HMI tags "2905RS001A01F02"
   "2905RS001A01F02.MSW" : 52809b66-421d-457f-8884-6f7a49d4e247 AT %DB5024.DBX18.0, 500 ms
   "2905RS001A01F02.DefaultText" : TextRef, internal   // Заголовок POPUP окна. При експорте из ECS через скрипт заполняется автоматически, если теги копируются в ручную то требуется в ручную задатать свойство Start Value
   "2905RS001A01F02.BlockInfo" : Array [0..2] of Int AT %DB5024.DBX38.0, 500 ms
   "2905RS001A01F02.StatusWork" : Int AT %DB5024.DBW242, 500 ms
   "2905RS001A01F02.FP_PARAM.DampingTime" : Int AT %DB5024.DBW50, 500 ms
   "2905RS001A01F02.FP_PARAM.Force_Value" : Real AT %DB5024.DBD52, 500 ms
   "2905RS001A01F02.FP_PARAM.Scale_Min" : Real AT %DB5024.DBD56, 500 ms
   "2905RS001A01F02.FP_PARAM.Scale_Max" : Real AT %DB5024.DBD60, 500 ms
   "2905RS001A01F02.FP_PARAM.Gradient" : Real AT %DB5024.DBD64, 500 ms
   "2905RS001A01F02.FP_PARAM.Grad_Pos" : Real AT %DB5024.DBD68, 500 ms
   "2905RS001A01F02.FP_PARAM.Grad_Neg" : Real AT %DB5024.DBD72, 500 ms
   "2905RS001A01F02.FP_PARAM.Grad_X" : Real AT %DB5024.DBD76, 500 ms
   "2905RS001A01F02.FP_PARAM.Gradient_Time_Pre" : Int AT %DB5024.DBW80, 500 ms
   "2905RS001A01F02.FP_PARAM.Gradient_Time_ACC" : Int AT %DB5024.DBW82, 500 ms
   "2905RS001A01F02.FP_PARAM.Alarm_Hyst" : Real AT %DB5024.DBD84, 500 ms
   "2905RS001A01F02.FP_PARAM.AlarmLimit_H3" : Real AT %DB5024.DBD88, 500 ms
   "2905RS001A01F02.FP_PARAM.AlarmLimit_H2" : Real AT %DB5024.DBD92, 500 ms
   "2905RS001A01F02.FP_PARAM.AlarmLimit_H1" : Real AT %DB5024.DBD96, 500 ms
   "2905RS001A01F02.FP_PARAM.AlarmLimit_L1" : Real AT %DB5024.DBD100, 500 ms
   "2905RS001A01F02.FP_PARAM.AlarmLimit_L2" : Real AT %DB5024.DBD104, 500 ms
   "2905RS001A01F02.FP_PARAM.AlarmLimit_L3" : Real AT %DB5024.DBD108, 500 ms
   "2905RS001A01F02.FP_PARAM.AlarmDelay_H3_Pre" : Int AT %DB5024.DBW112, 500 ms
   "2905RS001A01F02.FP_PARAM.AlarmDelay_H3_Acc" : Int AT %DB5024.DBW114, 500 ms
   "2905RS001A01F02.FP_PARAM.AlarmDelay_H2_Pre" : Int AT %DB5024.DBW116, 500 ms
   "2905RS001A01F02.FP_PARAM.AlarmDelay_H2_Acc" : Int AT %DB5024.DBW118, 500 ms
   "2905RS001A01F02.FP_PARAM.AlarmDelay_H1_Pre" : Int AT %DB5024.DBW120, 500 ms
   "2905RS001A01F02.FP_PARAM.AlarmDelay_H1_Acc" : Int AT %DB5024.DBW122, 500 ms
   "2905RS001A01F02.FP_PARAM.AlarmDelay_L1_Pre" : Int AT %DB5024.DBW124, 500 ms
   "2905RS001A01F02.FP_PARAM.AlarmDelay_L1_Acc" : Int AT %DB5024.DBW126, 500 ms
   "2905RS001A01F02.FP_PARAM.AlarmDelay_L2_Pre" : Int AT %DB5024.DBW128, 500 ms
   "2905RS001A01F02.FP_PARAM.AlarmDelay_L2_Acc" : Int AT %DB5024.DBW130, 500 ms
   "2905RS001A01F02.FP_PARAM.AlarmDelay_L3_Pre" : Int AT %DB5024.DBW132, 500 ms
   "2905RS001A01F02.FP_PARAM.AlarmDelay_L3_Acc" : Int AT %DB5024.DBW134, 500 ms
   "2905RS001A01F02.FP_PARAM.OpenLoopDelay_Pre" : Int AT %DB5024.DBW136, 500 ms
   "2905RS001A01F02.FP_PARAM.OpenLoopDelay_Acc" : Int AT %DB5024.DBW138, 500 ms
   "2905RS001A01F02.FP_PARAM.OverRangeDelay_Pre" : Int AT %DB5024.DBW140, 500 ms
   "2905RS001A01F02.FP_PARAM.OverRangeDelay_Acc" : Int AT %DB5024.DBW142, 500 ms
   "2905RS001A01F02.FP_PARAM.AuxLimit_H2_Value" : Real AT %DB5024.DBD144, 500 ms
   "2905RS001A01F02.FP_PARAM.AuxLimit_H1_Value" : Real AT %DB5024.DBD148, 500 ms
   "2905RS001A01F02.FP_PARAM.AuxLimit_L2_Value" : Real AT %DB5024.DBD152, 500 ms
   "2905RS001A01F02.FP_PARAM.AuxLimit_L1_Value" : Real AT %DB5024.DBD156, 500 ms
   "2905RS001A01F02.Unit" : TextRef, internal   // Еденицы измерения При експорте из ECS через скрипт заполняется автоматически, если теги копируются в ручную то требуется задатать свойство Text
   "2905RS001A01F02.Decimals" : TextRef, internal   // Формат отображения При експорте из ECS через скрипт, заполняется автоматически. Если теги копируются в ручную то требуется задатать свойство Text s999999.9
   "2905RS001A01F02.FP_EN.Square" : Bool AT %DB5024.DBX46.0, 500 ms
   "2905RS001A01F02.FP_EN.SquareRoot" : Bool AT %DB5024.DBX46.1, 500 ms
   "2905RS001A01F02.FP_EN.ParentSupress" : Bool AT %DB5024.DBX46.2, 500 ms
   "2905RS001A01F02.FP_EN.ParentSupressUnit" : Bool AT %DB5024.DBX46.3, 500 ms
   "2905RS001A01F02.FP_EN.Force" : Bool AT %DB5024.DBX46.4, 500 ms
   "2905RS001A01F02.FP_EN.Damping" : Bool AT %DB5024.DBX46.5, 500 ms
   "2905RS001A01F02.FP_EN.Gradient_Pos" : Bool AT %DB5024.DBX46.6, 500 ms
   "2905RS001A01F02.FP_EN.Gradient_Neg" : Bool AT %DB5024.DBX46.7, 500 ms
   "2905RS001A01F02.FP_EN.Hysteresis" : Bool AT %DB5024.DBX47.0, 500 ms
   "2905RS001A01F02.FP_EN.Alarm_H3" : Bool AT %DB5024.DBX47.1, 500 ms
   "2905RS001A01F02.FP_EN.Alarm_H2" : Bool AT %DB5024.DBX47.2, 500 ms
   "2905RS001A01F02.FP_EN.Alarm_H1" : Bool AT %DB5024.DBX47.3, 500 ms
   "2905RS001A01F02.FP_EN.Alarm_L1" : Bool AT %DB5024.DBX47.4, 500 ms
   "2905RS001A01F02.FP_EN.Alarm_L2" : Bool AT %DB5024.DBX47.5, 500 ms
   "2905RS001A01F02.FP_EN.Alarm_L3" : Bool AT %DB5024.DBX47.6, 500 ms
   "2905RS001A01F02.FP_EN.AlarmDelay_H3" : Bool AT %DB5024.DBX47.7, 500 ms
   "2905RS001A01F02.FP_EN.AlarmDelay_H2" : Bool AT %DB5024.DBX48.0, 500 ms
   "2905RS001A01F02.FP_EN.AlarmDelay_H1" : Bool AT %DB5024.DBX48.1, 500 ms
   "2905RS001A01F02.FP_EN.AlarmDelay_L1" : Bool AT %DB5024.DBX48.2, 500 ms
   "2905RS001A01F02.FP_EN.AlarmDelay_L2" : Bool AT %DB5024.DBX48.3, 500 ms
   "2905RS001A01F02.FP_EN.AlarmDelay_L3" : Bool AT %DB5024.DBX48.4, 500 ms
   "2905RS001A01F02.FP_EN.ROC_Warn" : Bool AT %DB5024.DBX48.5, 500 ms
   "2905RS001A01F02.FP_EN.U_Range_Warn" : Bool AT %DB5024.DBX48.6, 500 ms
   "2905RS001A01F02.FP_EN.O_Range_Warn" : Bool AT %DB5024.DBX48.7, 500 ms
   "2905RS001A01F02.trend_tag_name" : TextRef, internal   // Еденицы измерения При експорте из ECS через скрипт - заполняется автоматически, если теги копируются в ручную то требуется задатать свойство Text - имя тега для тренда
   "2905RS001A01F02.DQ.AL_H3" : Bool AT %DB5024.DBX16.0, 500 ms
   "2905RS001A01F02.DQ.AL_H2" : Bool AT %DB5024.DBX16.1, 500 ms
   "2905RS001A01F02.DQ.AL_H1" : Bool AT %DB5024.DBX16.2, 500 ms
   "2905RS001A01F02.DQ.AL_L1" : Bool AT %DB5024.DBX16.3, 500 ms
   "2905RS001A01F02.DQ.AL_L2" : Bool AT %DB5024.DBX16.4, 500 ms
   "2905RS001A01F02.DQ.AL_L3" : Bool AT %DB5024.DBX16.5, 500 ms
   "2905RS001A01F02.DQ.SIG_OK" : Bool AT %DB5024.DBX16.6, 500 ms
   "2905RS001A01F02.DQ.LIM_H2" : Bool AT %DB5024.DBX16.7, 500 ms
   "2905RS001A01F02.DQ.LIM_H1" : Bool AT %DB5024.DBX17.0, 500 ms
   "2905RS001A01F02.DQ.LIM_L1" : Bool AT %DB5024.DBX17.1, 500 ms
   "2905RS001A01F02.DQ.LIM_L2" : Bool AT %DB5024.DBX17.2, 500 ms
   "2905RS001A01F02.DQ.GR_P" : Bool AT %DB5024.DBX17.3, 500 ms
   "2905RS001A01F02.DQ.GR_N" : Bool AT %DB5024.DBX17.4, 500 ms
   "2905RS001A01F02.I.IN" : Real AT %DB5024.DBD2, 500 ms
   "2905RS001A01F02.I.SIG_TYPE" : Int AT %DB5024.DBW0, 500 ms
   "2905RS001A01F02.I.FI_BUS" : Byte AT %DB5024.DBB6, 500 ms
   "2905RS001A01F02.DI.U_RANGE" : Bool AT %DB5024.DBX7.0, 500 ms
   "2905RS001A01F02.DI.O_RANGE" : Bool AT %DB5024.DBX7.1, 500 ms
   "2905RS001A01F02.DI.SIG_FAULT" : Bool AT %DB5024.DBX7.2, 500 ms
   "2905RS001A01F02.DI.EnConfig" : Bool AT %DB5024.DBX7.3, 500 ms
   "2905RS001A01F02.DI.AEN" : Bool AT %DB5024.DBX7.4, 500 ms
   "2905RS001A01F02.DI.AL_SUPR" : Bool AT %DB5024.DBX7.5, 500 ms
   "2905RS001A01F02.Q.PV_NORM" : Real AT %DB5024.DBD8, 500 ms
   "2905RS001A01F02.Q.PV_SCAL" : Real AT %DB5024.DBD12, 500 ms
   "2905RS001A01F02.ParentInfo" : TextRef, internal   // Имя родителя для попап окна, вкладка инфо. При експорте из ECS через скрипт заполняется автоматически, если теги копируются в ручную то требуется в ручную задатать свойство Start Value

HMI tags "2905RS001A01F03"
   "2905RS001A01F03.MSW" : 52809b66-421d-457f-8884-6f7a49d4e247 AT %DB5025.DBX18.0, 500 ms
   "2905RS001A01F03.DefaultText" : TextRef, internal   // Заголовок POPUP окна. При експорте из ECS через скрипт заполняется автоматически, если теги копируются в ручную то требуется в ручную задатать свойство Start Value
   "2905RS001A01F03.BlockInfo" : Array [0..2] of Int AT %DB5025.DBX38.0, 500 ms
   "2905RS001A01F03.StatusWork" : Int AT %DB5025.DBW242, 500 ms
   "2905RS001A01F03.FP_PARAM.DampingTime" : Int AT %DB5025.DBW50, 500 ms
   "2905RS001A01F03.FP_PARAM.Force_Value" : Real AT %DB5025.DBD52, 500 ms
   "2905RS001A01F03.FP_PARAM.Scale_Min" : Real AT %DB5025.DBD56, 500 ms
   "2905RS001A01F03.FP_PARAM.Scale_Max" : Real AT %DB5025.DBD60, 500 ms
   "2905RS001A01F03.FP_PARAM.Gradient" : Real AT %DB5025.DBD64, 500 ms
   "2905RS001A01F03.FP_PARAM.Grad_Pos" : Real AT %DB5025.DBD68, 500 ms
   "2905RS001A01F03.FP_PARAM.Grad_Neg" : Real AT %DB5025.DBD72, 500 ms
   "2905RS001A01F03.FP_PARAM.Grad_X" : Real AT %DB5025.DBD76, 500 ms
   "2905RS001A01F03.FP_PARAM.Gradient_Time_Pre" : Int AT %DB5025.DBW80, 500 ms
   "2905RS001A01F03.FP_PARAM.Gradient_Time_ACC" : Int AT %DB5025.DBW82, 500 ms
   "2905RS001A01F03.FP_PARAM.Alarm_Hyst" : Real AT %DB5025.DBD84, 500 ms
   "2905RS001A01F03.FP_PARAM.AlarmLimit_H3" : Real AT %DB5025.DBD88, 500 ms
   "2905RS001A01F03.FP_PARAM.AlarmLimit_H2" : Real AT %DB5025.DBD92, 500 ms
   "2905RS001A01F03.FP_PARAM.AlarmLimit_H1" : Real AT %DB5025.DBD96, 500 ms
   "2905RS001A01F03.FP_PARAM.AlarmLimit_L1" : Real AT %DB5025.DBD100, 500 ms
   "2905RS001A01F03.FP_PARAM.AlarmLimit_L2" : Real AT %DB5025.DBD104, 500 ms
   "2905RS001A01F03.FP_PARAM.AlarmLimit_L3" : Real AT %DB5025.DBD108, 500 ms
   "2905RS001A01F03.FP_PARAM.AlarmDelay_H3_Pre" : Int AT %DB5025.DBW112, 500 ms
   "2905RS001A01F03.FP_PARAM.AlarmDelay_H3_Acc" : Int AT %DB5025.DBW114, 500 ms
   "2905RS001A01F03.FP_PARAM.AlarmDelay_H2_Pre" : Int AT %DB5025.DBW116, 500 ms
   "2905RS001A01F03.FP_PARAM.AlarmDelay_H2_Acc" : Int AT %DB5025.DBW118, 500 ms
   "2905RS001A01F03.FP_PARAM.AlarmDelay_H1_Pre" : Int AT %DB5025.DBW120, 500 ms
   "2905RS001A01F03.FP_PARAM.AlarmDelay_H1_Acc" : Int AT %DB5025.DBW122, 500 ms
   "2905RS001A01F03.FP_PARAM.AlarmDelay_L1_Pre" : Int AT %DB5025.DBW124, 500 ms
   "2905RS001A01F03.FP_PARAM.AlarmDelay_L1_Acc" : Int AT %DB5025.DBW126, 500 ms
   "2905RS001A01F03.FP_PARAM.AlarmDelay_L2_Pre" : Int AT %DB5025.DBW128, 500 ms
   "2905RS001A01F03.FP_PARAM.AlarmDelay_L2_Acc" : Int AT %DB5025.DBW130, 500 ms
   "2905RS001A01F03.FP_PARAM.AlarmDelay_L3_Pre" : Int AT %DB5025.DBW132, 500 ms
   "2905RS001A01F03.FP_PARAM.AlarmDelay_L3_Acc" : Int AT %DB5025.DBW134, 500 ms
   "2905RS001A01F03.FP_PARAM.OpenLoopDelay_Pre" : Int AT %DB5025.DBW136, 500 ms
   "2905RS001A01F03.FP_PARAM.OpenLoopDelay_Acc" : Int AT %DB5025.DBW138, 500 ms
   "2905RS001A01F03.FP_PARAM.OverRangeDelay_Pre" : Int AT %DB5025.DBW140, 500 ms
   "2905RS001A01F03.FP_PARAM.OverRangeDelay_Acc" : Int AT %DB5025.DBW142, 500 ms
   "2905RS001A01F03.FP_PARAM.AuxLimit_H2_Value" : Real AT %DB5025.DBD144, 500 ms
   "2905RS001A01F03.FP_PARAM.AuxLimit_H1_Value" : Real AT %DB5025.DBD148, 500 ms
   "2905RS001A01F03.FP_PARAM.AuxLimit_L2_Value" : Real AT %DB5025.DBD152, 500 ms
   "2905RS001A01F03.FP_PARAM.AuxLimit_L1_Value" : Real AT %DB5025.DBD156, 500 ms
   "2905RS001A01F03.Unit" : TextRef, internal   // Еденицы измерения При експорте из ECS через скрипт заполняется автоматически, если теги копируются в ручную то требуется задатать свойство Text
   "2905RS001A01F03.Decimals" : TextRef, internal   // Формат отображения При експорте из ECS через скрипт, заполняется автоматически. Если теги копируются в ручную то требуется задатать свойство Text s999999.9
   "2905RS001A01F03.FP_EN.Square" : Bool AT %DB5025.DBX46.0, 500 ms
   "2905RS001A01F03.FP_EN.SquareRoot" : Bool AT %DB5025.DBX46.1, 500 ms
   "2905RS001A01F03.FP_EN.ParentSupress" : Bool AT %DB5025.DBX46.2, 500 ms
   "2905RS001A01F03.FP_EN.ParentSupressUnit" : Bool AT %DB5025.DBX46.3, 500 ms
   "2905RS001A01F03.FP_EN.Force" : Bool AT %DB5025.DBX46.4, 500 ms
   "2905RS001A01F03.FP_EN.Damping" : Bool AT %DB5025.DBX46.5, 500 ms
   "2905RS001A01F03.FP_EN.Gradient_Pos" : Bool AT %DB5025.DBX46.6, 500 ms
   "2905RS001A01F03.FP_EN.Gradient_Neg" : Bool AT %DB5025.DBX46.7, 500 ms
   "2905RS001A01F03.FP_EN.Hysteresis" : Bool AT %DB5025.DBX47.0, 500 ms
   "2905RS001A01F03.FP_EN.Alarm_H3" : Bool AT %DB5025.DBX47.1, 500 ms
   "2905RS001A01F03.FP_EN.Alarm_H2" : Bool AT %DB5025.DBX47.2, 500 ms
   "2905RS001A01F03.FP_EN.Alarm_H1" : Bool AT %DB5025.DBX47.3, 500 ms
   "2905RS001A01F03.FP_EN.Alarm_L1" : Bool AT %DB5025.DBX47.4, 500 ms
   "2905RS001A01F03.FP_EN.Alarm_L2" : Bool AT %DB5025.DBX47.5, 500 ms
   "2905RS001A01F03.FP_EN.Alarm_L3" : Bool AT %DB5025.DBX47.6, 500 ms
   "2905RS001A01F03.FP_EN.AlarmDelay_H3" : Bool AT %DB5025.DBX47.7, 500 ms
   "2905RS001A01F03.FP_EN.AlarmDelay_H2" : Bool AT %DB5025.DBX48.0, 500 ms
   "2905RS001A01F03.FP_EN.AlarmDelay_H1" : Bool AT %DB5025.DBX48.1, 500 ms
   "2905RS001A01F03.FP_EN.AlarmDelay_L1" : Bool AT %DB5025.DBX48.2, 500 ms
   "2905RS001A01F03.FP_EN.AlarmDelay_L2" : Bool AT %DB5025.DBX48.3, 500 ms
   "2905RS001A01F03.FP_EN.AlarmDelay_L3" : Bool AT %DB5025.DBX48.4, 500 ms
   "2905RS001A01F03.FP_EN.ROC_Warn" : Bool AT %DB5025.DBX48.5, 500 ms
   "2905RS001A01F03.FP_EN.U_Range_Warn" : Bool AT %DB5025.DBX48.6, 500 ms
   "2905RS001A01F03.FP_EN.O_Range_Warn" : Bool AT %DB5025.DBX48.7, 500 ms
   "2905RS001A01F03.trend_tag_name" : TextRef, internal   // Еденицы измерения При експорте из ECS через скрипт - заполняется автоматически, если теги копируются в ручную то требуется задатать свойство Text - имя тега для тренда
   "2905RS001A01F03.DQ.AL_H3" : Bool AT %DB5025.DBX16.0, 500 ms
   "2905RS001A01F03.DQ.AL_H2" : Bool AT %DB5025.DBX16.1, 500 ms
   "2905RS001A01F03.DQ.AL_H1" : Bool AT %DB5025.DBX16.2, 500 ms
   "2905RS001A01F03.DQ.AL_L1" : Bool AT %DB5025.DBX16.3, 500 ms
   "2905RS001A01F03.DQ.AL_L2" : Bool AT %DB5025.DBX16.4, 500 ms
   "2905RS001A01F03.DQ.AL_L3" : Bool AT %DB5025.DBX16.5, 500 ms
   "2905RS001A01F03.DQ.SIG_OK" : Bool AT %DB5025.DBX16.6, 500 ms
   "2905RS001A01F03.DQ.LIM_H2" : Bool AT %DB5025.DBX16.7, 500 ms
   "2905RS001A01F03.DQ.LIM_H1" : Bool AT %DB5025.DBX17.0, 500 ms
   "2905RS001A01F03.DQ.LIM_L1" : Bool AT %DB5025.DBX17.1, 500 ms
   "2905RS001A01F03.DQ.LIM_L2" : Bool AT %DB5025.DBX17.2, 500 ms
   "2905RS001A01F03.DQ.GR_P" : Bool AT %DB5025.DBX17.3, 500 ms
   "2905RS001A01F03.DQ.GR_N" : Bool AT %DB5025.DBX17.4, 500 ms
   "2905RS001A01F03.I.IN" : Real AT %DB5025.DBD2, 500 ms
   "2905RS001A01F03.I.SIG_TYPE" : Int AT %DB5025.DBW0, 500 ms
   "2905RS001A01F03.I.FI_BUS" : Byte AT %DB5025.DBB6, 500 ms
   "2905RS001A01F03.DI.U_RANGE" : Bool AT %DB5025.DBX7.0, 500 ms
   "2905RS001A01F03.DI.O_RANGE" : Bool AT %DB5025.DBX7.1, 500 ms
   "2905RS001A01F03.DI.SIG_FAULT" : Bool AT %DB5025.DBX7.2, 500 ms
   "2905RS001A01F03.DI.EnConfig" : Bool AT %DB5025.DBX7.3, 500 ms
   "2905RS001A01F03.DI.AEN" : Bool AT %DB5025.DBX7.4, 500 ms
   "2905RS001A01F03.DI.AL_SUPR" : Bool AT %DB5025.DBX7.5, 500 ms
   "2905RS001A01F03.Q.PV_NORM" : Real AT %DB5025.DBD8, 500 ms
   "2905RS001A01F03.Q.PV_SCAL" : Real AT %DB5025.DBD12, 500 ms
   "2905RS001A01F03.ParentInfo" : TextRef, internal   // Имя родителя для попап окна, вкладка инфо. При експорте из ECS через скрипт заполняется автоматически, если теги копируются в ручную то требуется в ручную задатать свойство Start Value

HMI tags "2905RS001A01F04"
   "2905RS001A01F04.MSW" : 52809b66-421d-457f-8884-6f7a49d4e247 AT %DB5026.DBX18.0, 500 ms
   "2905RS001A01F04.DefaultText" : TextRef, internal   // Заголовок POPUP окна. При експорте из ECS через скрипт заполняется автоматически, если теги копируются в ручную то требуется в ручную задатать свойство Start Value
   "2905RS001A01F04.BlockInfo" : Array [0..2] of Int AT %DB5026.DBX38.0, 500 ms
   "2905RS001A01F04.StatusWork" : Int AT %DB5026.DBW242, 500 ms
   "2905RS001A01F04.FP_PARAM.DampingTime" : Int AT %DB5026.DBW50, 500 ms
   "2905RS001A01F04.FP_PARAM.Force_Value" : Real AT %DB5026.DBD52, 500 ms
   "2905RS001A01F04.FP_PARAM.Scale_Min" : Real AT %DB5026.DBD56, 500 ms
   "2905RS001A01F04.FP_PARAM.Scale_Max" : Real AT %DB5026.DBD60, 500 ms
   "2905RS001A01F04.FP_PARAM.Gradient" : Real AT %DB5026.DBD64, 500 ms
   "2905RS001A01F04.FP_PARAM.Grad_Pos" : Real AT %DB5026.DBD68, 500 ms
   "2905RS001A01F04.FP_PARAM.Grad_Neg" : Real AT %DB5026.DBD72, 500 ms
   "2905RS001A01F04.FP_PARAM.Grad_X" : Real AT %DB5026.DBD76, 500 ms
   "2905RS001A01F04.FP_PARAM.Gradient_Time_Pre" : Int AT %DB5026.DBW80, 500 ms
   "2905RS001A01F04.FP_PARAM.Gradient_Time_ACC" : Int AT %DB5026.DBW82, 500 ms
   "2905RS001A01F04.FP_PARAM.Alarm_Hyst" : Real AT %DB5026.DBD84, 500 ms
   "2905RS001A01F04.FP_PARAM.AlarmLimit_H3" : Real AT %DB5026.DBD88, 500 ms
   "2905RS001A01F04.FP_PARAM.AlarmLimit_H2" : Real AT %DB5026.DBD92, 500 ms
   "2905RS001A01F04.FP_PARAM.AlarmLimit_H1" : Real AT %DB5026.DBD96, 500 ms
   "2905RS001A01F04.FP_PARAM.AlarmLimit_L1" : Real AT %DB5026.DBD100, 500 ms
   "2905RS001A01F04.FP_PARAM.AlarmLimit_L2" : Real AT %DB5026.DBD104, 500 ms
   "2905RS001A01F04.FP_PARAM.AlarmLimit_L3" : Real AT %DB5026.DBD108, 500 ms
   "2905RS001A01F04.FP_PARAM.AlarmDelay_H3_Pre" : Int AT %DB5026.DBW112, 500 ms
   "2905RS001A01F04.FP_PARAM.AlarmDelay_H3_Acc" : Int AT %DB5026.DBW114, 500 ms
   "2905RS001A01F04.FP_PARAM.AlarmDelay_H2_Pre" : Int AT %DB5026.DBW116, 500 ms
   "2905RS001A01F04.FP_PARAM.AlarmDelay_H2_Acc" : Int AT %DB5026.DBW118, 500 ms
   "2905RS001A01F04.FP_PARAM.AlarmDelay_H1_Pre" : Int AT %DB5026.DBW120, 500 ms
   "2905RS001A01F04.FP_PARAM.AlarmDelay_H1_Acc" : Int AT %DB5026.DBW122, 500 ms
   "2905RS001A01F04.FP_PARAM.AlarmDelay_L1_Pre" : Int AT %DB5026.DBW124, 500 ms
   "2905RS001A01F04.FP_PARAM.AlarmDelay_L1_Acc" : Int AT %DB5026.DBW126, 500 ms
   "2905RS001A01F04.FP_PARAM.AlarmDelay_L2_Pre" : Int AT %DB5026.DBW128, 500 ms
   "2905RS001A01F04.FP_PARAM.AlarmDelay_L2_Acc" : Int AT %DB5026.DBW130, 500 ms
   "2905RS001A01F04.FP_PARAM.AlarmDelay_L3_Pre" : Int AT %DB5026.DBW132, 500 ms
   "2905RS001A01F04.FP_PARAM.AlarmDelay_L3_Acc" : Int AT %DB5026.DBW134, 500 ms
   "2905RS001A01F04.FP_PARAM.OpenLoopDelay_Pre" : Int AT %DB5026.DBW136, 500 ms
   "2905RS001A01F04.FP_PARAM.OpenLoopDelay_Acc" : Int AT %DB5026.DBW138, 500 ms
   "2905RS001A01F04.FP_PARAM.OverRangeDelay_Pre" : Int AT %DB5026.DBW140, 500 ms
   "2905RS001A01F04.FP_PARAM.OverRangeDelay_Acc" : Int AT %DB5026.DBW142, 500 ms
   "2905RS001A01F04.FP_PARAM.AuxLimit_H2_Value" : Real AT %DB5026.DBD144, 500 ms
   "2905RS001A01F04.FP_PARAM.AuxLimit_H1_Value" : Real AT %DB5026.DBD148, 500 ms
   "2905RS001A01F04.FP_PARAM.AuxLimit_L2_Value" : Real AT %DB5026.DBD152, 500 ms
   "2905RS001A01F04.FP_PARAM.AuxLimit_L1_Value" : Real AT %DB5026.DBD156, 500 ms
   "2905RS001A01F04.Unit" : TextRef, internal   // Еденицы измерения При експорте из ECS через скрипт заполняется автоматически, если теги копируются в ручную то требуется задатать свойство Text
   "2905RS001A01F04.Decimals" : TextRef, internal   // Формат отображения При експорте из ECS через скрипт, заполняется автоматически. Если теги копируются в ручную то требуется задатать свойство Text s999999.9
   "2905RS001A01F04.FP_EN.Square" : Bool AT %DB5026.DBX46.0, 500 ms
   "2905RS001A01F04.FP_EN.SquareRoot" : Bool AT %DB5026.DBX46.1, 500 ms
   "2905RS001A01F04.FP_EN.ParentSupress" : Bool AT %DB5026.DBX46.2, 500 ms
   "2905RS001A01F04.FP_EN.ParentSupressUnit" : Bool AT %DB5026.DBX46.3, 500 ms
   "2905RS001A01F04.FP_EN.Force" : Bool AT %DB5026.DBX46.4, 500 ms
   "2905RS001A01F04.FP_EN.Damping" : Bool AT %DB5026.DBX46.5, 500 ms
   "2905RS001A01F04.FP_EN.Gradient_Pos" : Bool AT %DB5026.DBX46.6, 500 ms
   "2905RS001A01F04.FP_EN.Gradient_Neg" : Bool AT %DB5026.DBX46.7, 500 ms
   "2905RS001A01F04.FP_EN.Hysteresis" : Bool AT %DB5026.DBX47.0, 500 ms
   "2905RS001A01F04.FP_EN.Alarm_H3" : Bool AT %DB5026.DBX47.1, 500 ms
   "2905RS001A01F04.FP_EN.Alarm_H2" : Bool AT %DB5026.DBX47.2, 500 ms
   "2905RS001A01F04.FP_EN.Alarm_H1" : Bool AT %DB5026.DBX47.3, 500 ms
   "2905RS001A01F04.FP_EN.Alarm_L1" : Bool AT %DB5026.DBX47.4, 500 ms
   "2905RS001A01F04.FP_EN.Alarm_L2" : Bool AT %DB5026.DBX47.5, 500 ms
   "2905RS001A01F04.FP_EN.Alarm_L3" : Bool AT %DB5026.DBX47.6, 500 ms
   "2905RS001A01F04.FP_EN.AlarmDelay_H3" : Bool AT %DB5026.DBX47.7, 500 ms
   "2905RS001A01F04.FP_EN.AlarmDelay_H2" : Bool AT %DB5026.DBX48.0, 500 ms
   "2905RS001A01F04.FP_EN.AlarmDelay_H1" : Bool AT %DB5026.DBX48.1, 500 ms
   "2905RS001A01F04.FP_EN.AlarmDelay_L1" : Bool AT %DB5026.DBX48.2, 500 ms
   "2905RS001A01F04.FP_EN.AlarmDelay_L2" : Bool AT %DB5026.DBX48.3, 500 ms
   "2905RS001A01F04.FP_EN.AlarmDelay_L3" : Bool AT %DB5026.DBX48.4, 500 ms
   "2905RS001A01F04.FP_EN.ROC_Warn" : Bool AT %DB5026.DBX48.5, 500 ms
   "2905RS001A01F04.FP_EN.U_Range_Warn" : Bool AT %DB5026.DBX48.6, 500 ms
   "2905RS001A01F04.FP_EN.O_Range_Warn" : Bool AT %DB5026.DBX48.7, 500 ms
   "2905RS001A01F04.trend_tag_name" : TextRef, internal   // Еденицы измерения При експорте из ECS через скрипт - заполняется автоматически, если теги копируются в ручную то требуется задатать свойство Text - имя тега для тренда
   "2905RS001A01F04.DQ.AL_H3" : Bool AT %DB5026.DBX16.0, 500 ms
   "2905RS001A01F04.DQ.AL_H2" : Bool AT %DB5026.DBX16.1, 500 ms
   "2905RS001A01F04.DQ.AL_H1" : Bool AT %DB5026.DBX16.2, 500 ms
   "2905RS001A01F04.DQ.AL_L1" : Bool AT %DB5026.DBX16.3, 500 ms
   "2905RS001A01F04.DQ.AL_L2" : Bool AT %DB5026.DBX16.4, 500 ms
   "2905RS001A01F04.DQ.AL_L3" : Bool AT %DB5026.DBX16.5, 500 ms
   "2905RS001A01F04.DQ.SIG_OK" : Bool AT %DB5026.DBX16.6, 500 ms
   "2905RS001A01F04.DQ.LIM_H2" : Bool AT %DB5026.DBX16.7, 500 ms
   "2905RS001A01F04.DQ.LIM_H1" : Bool AT %DB5026.DBX17.0, 500 ms
   "2905RS001A01F04.DQ.LIM_L1" : Bool AT %DB5026.DBX17.1, 500 ms
   "2905RS001A01F04.DQ.LIM_L2" : Bool AT %DB5026.DBX17.2, 500 ms
   "2905RS001A01F04.DQ.GR_P" : Bool AT %DB5026.DBX17.3, 500 ms
   "2905RS001A01F04.DQ.GR_N" : Bool AT %DB5026.DBX17.4, 500 ms
   "2905RS001A01F04.I.IN" : Real AT %DB5026.DBD2, 500 ms
   "2905RS001A01F04.I.SIG_TYPE" : Int AT %DB5026.DBW0, 500 ms
   "2905RS001A01F04.I.FI_BUS" : Byte AT %DB5026.DBB6, 500 ms
   "2905RS001A01F04.DI.U_RANGE" : Bool AT %DB5026.DBX7.0, 500 ms
   "2905RS001A01F04.DI.O_RANGE" : Bool AT %DB5026.DBX7.1, 500 ms
   "2905RS001A01F04.DI.SIG_FAULT" : Bool AT %DB5026.DBX7.2, 500 ms
   "2905RS001A01F04.DI.EnConfig" : Bool AT %DB5026.DBX7.3, 500 ms
   "2905RS001A01F04.DI.AEN" : Bool AT %DB5026.DBX7.4, 500 ms
   "2905RS001A01F04.DI.AL_SUPR" : Bool AT %DB5026.DBX7.5, 500 ms
   "2905RS001A01F04.Q.PV_NORM" : Real AT %DB5026.DBD8, 500 ms
   "2905RS001A01F04.Q.PV_SCAL" : Real AT %DB5026.DBD12, 500 ms
   "2905RS001A01F04.ParentInfo" : TextRef, internal   // Имя родителя для попап окна, вкладка инфо. При експорте из ECS через скрипт заполняется автоматически, если теги копируются в ручную то требуется в ручную задатать свойство Start Value

HMI tags "2905RS001A01L01"
   "2905RS001A01L01.MSW" : 52809b66-421d-457f-8884-6f7a49d4e247 AT %DB5027.DBX18.0, 500 ms
   "2905RS001A01L01.DefaultText" : TextRef, internal   // Заголовок POPUP окна. При експорте из ECS через скрипт заполняется автоматически, если теги копируются в ручную то требуется в ручную задатать свойство Start Value
   "2905RS001A01L01.BlockInfo" : Array [0..2] of Int AT %DB5027.DBX38.0, 500 ms
   "2905RS001A01L01.StatusWork" : Int AT %DB5027.DBW242, 500 ms
   "2905RS001A01L01.FP_PARAM.DampingTime" : Int AT %DB5027.DBW50, 500 ms
   "2905RS001A01L01.FP_PARAM.Force_Value" : Real AT %DB5027.DBD52, 500 ms
   "2905RS001A01L01.FP_PARAM.Scale_Min" : Real AT %DB5027.DBD56, 500 ms
   "2905RS001A01L01.FP_PARAM.Scale_Max" : Real AT %DB5027.DBD60, 500 ms
   "2905RS001A01L01.FP_PARAM.Gradient" : Real AT %DB5027.DBD64, 500 ms
   "2905RS001A01L01.FP_PARAM.Grad_Pos" : Real AT %DB5027.DBD68, 500 ms
   "2905RS001A01L01.FP_PARAM.Grad_Neg" : Real AT %DB5027.DBD72, 500 ms
   "2905RS001A01L01.FP_PARAM.Grad_X" : Real AT %DB5027.DBD76, 500 ms
   "2905RS001A01L01.FP_PARAM.Gradient_Time_Pre" : Int AT %DB5027.DBW80, 500 ms
   "2905RS001A01L01.FP_PARAM.Gradient_Time_ACC" : Int AT %DB5027.DBW82, 500 ms
   "2905RS001A01L01.FP_PARAM.Alarm_Hyst" : Real AT %DB5027.DBD84, 500 ms
   "2905RS001A01L01.FP_PARAM.AlarmLimit_H3" : Real AT %DB5027.DBD88, 500 ms
   "2905RS001A01L01.FP_PARAM.AlarmLimit_H2" : Real AT %DB5027.DBD92, 500 ms
   "2905RS001A01L01.FP_PARAM.AlarmLimit_H1" : Real AT %DB5027.DBD96, 500 ms
   "2905RS001A01L01.FP_PARAM.AlarmLimit_L1" : Real AT %DB5027.DBD100, 500 ms
   "2905RS001A01L01.FP_PARAM.AlarmLimit_L2" : Real AT %DB5027.DBD104, 500 ms
   "2905RS001A01L01.FP_PARAM.AlarmLimit_L3" : Real AT %DB5027.DBD108, 500 ms
   "2905RS001A01L01.FP_PARAM.AlarmDelay_H3_Pre" : Int AT %DB5027.DBW112, 500 ms
   "2905RS001A01L01.FP_PARAM.AlarmDelay_H3_Acc" : Int AT %DB5027.DBW114, 500 ms
   "2905RS001A01L01.FP_PARAM.AlarmDelay_H2_Pre" : Int AT %DB5027.DBW116, 500 ms
   "2905RS001A01L01.FP_PARAM.AlarmDelay_H2_Acc" : Int AT %DB5027.DBW118, 500 ms
   "2905RS001A01L01.FP_PARAM.AlarmDelay_H1_Pre" : Int AT %DB5027.DBW120, 500 ms
   "2905RS001A01L01.FP_PARAM.AlarmDelay_H1_Acc" : Int AT %DB5027.DBW122, 500 ms
   "2905RS001A01L01.FP_PARAM.AlarmDelay_L1_Pre" : Int AT %DB5027.DBW124, 500 ms
   "2905RS001A01L01.FP_PARAM.AlarmDelay_L1_Acc" : Int AT %DB5027.DBW126, 500 ms
   "2905RS001A01L01.FP_PARAM.AlarmDelay_L2_Pre" : Int AT %DB5027.DBW128, 500 ms
   "2905RS001A01L01.FP_PARAM.AlarmDelay_L2_Acc" : Int AT %DB5027.DBW130, 500 ms
   "2905RS001A01L01.FP_PARAM.AlarmDelay_L3_Pre" : Int AT %DB5027.DBW132, 500 ms
   "2905RS001A01L01.FP_PARAM.AlarmDelay_L3_Acc" : Int AT %DB5027.DBW134, 500 ms
   "2905RS001A01L01.FP_PARAM.OpenLoopDelay_Pre" : Int AT %DB5027.DBW136, 500 ms
   "2905RS001A01L01.FP_PARAM.OpenLoopDelay_Acc" : Int AT %DB5027.DBW138, 500 ms
   "2905RS001A01L01.FP_PARAM.OverRangeDelay_Pre" : Int AT %DB5027.DBW140, 500 ms
   "2905RS001A01L01.FP_PARAM.OverRangeDelay_Acc" : Int AT %DB5027.DBW142, 500 ms
   "2905RS001A01L01.FP_PARAM.AuxLimit_H2_Value" : Real AT %DB5027.DBD144, 500 ms
   "2905RS001A01L01.FP_PARAM.AuxLimit_H1_Value" : Real AT %DB5027.DBD148, 500 ms
   "2905RS001A01L01.FP_PARAM.AuxLimit_L2_Value" : Real AT %DB5027.DBD152, 500 ms
   "2905RS001A01L01.FP_PARAM.AuxLimit_L1_Value" : Real AT %DB5027.DBD156, 500 ms
   "2905RS001A01L01.Unit" : TextRef, internal   // Еденицы измерения При експорте из ECS через скрипт заполняется автоматически, если теги копируются в ручную то требуется задатать свойство Text
   "2905RS001A01L01.Decimals" : TextRef, internal   // Формат отображения При експорте из ECS через скрипт, заполняется автоматически. Если теги копируются в ручную то требуется задатать свойство Text s999999.9
   "2905RS001A01L01.FP_EN.Square" : Bool AT %DB5027.DBX46.0, 500 ms
   "2905RS001A01L01.FP_EN.SquareRoot" : Bool AT %DB5027.DBX46.1, 500 ms
   "2905RS001A01L01.FP_EN.ParentSupress" : Bool AT %DB5027.DBX46.2, 500 ms
   "2905RS001A01L01.FP_EN.ParentSupressUnit" : Bool AT %DB5027.DBX46.3, 500 ms
   "2905RS001A01L01.FP_EN.Force" : Bool AT %DB5027.DBX46.4, 500 ms
   "2905RS001A01L01.FP_EN.Damping" : Bool AT %DB5027.DBX46.5, 500 ms
   "2905RS001A01L01.FP_EN.Gradient_Pos" : Bool AT %DB5027.DBX46.6, 500 ms
   "2905RS001A01L01.FP_EN.Gradient_Neg" : Bool AT %DB5027.DBX46.7, 500 ms
   "2905RS001A01L01.FP_EN.Hysteresis" : Bool AT %DB5027.DBX47.0, 500 ms
   "2905RS001A01L01.FP_EN.Alarm_H3" : Bool AT %DB5027.DBX47.1, 500 ms
   "2905RS001A01L01.FP_EN.Alarm_H2" : Bool AT %DB5027.DBX47.2, 500 ms
   "2905RS001A01L01.FP_EN.Alarm_H1" : Bool AT %DB5027.DBX47.3, 500 ms
   "2905RS001A01L01.FP_EN.Alarm_L1" : Bool AT %DB5027.DBX47.4, 500 ms
   "2905RS001A01L01.FP_EN.Alarm_L2" : Bool AT %DB5027.DBX47.5, 500 ms
   "2905RS001A01L01.FP_EN.Alarm_L3" : Bool AT %DB5027.DBX47.6, 500 ms
   "2905RS001A01L01.FP_EN.AlarmDelay_H3" : Bool AT %DB5027.DBX47.7, 500 ms
   "2905RS001A01L01.FP_EN.AlarmDelay_H2" : Bool AT %DB5027.DBX48.0, 500 ms
   "2905RS001A01L01.FP_EN.AlarmDelay_H1" : Bool AT %DB5027.DBX48.1, 500 ms
   "2905RS001A01L01.FP_EN.AlarmDelay_L1" : Bool AT %DB5027.DBX48.2, 500 ms
   "2905RS001A01L01.FP_EN.AlarmDelay_L2" : Bool AT %DB5027.DBX48.3, 500 ms
   "2905RS001A01L01.FP_EN.AlarmDelay_L3" : Bool AT %DB5027.DBX48.4, 500 ms
   "2905RS001A01L01.FP_EN.ROC_Warn" : Bool AT %DB5027.DBX48.5, 500 ms
   "2905RS001A01L01.FP_EN.U_Range_Warn" : Bool AT %DB5027.DBX48.6, 500 ms
   "2905RS001A01L01.FP_EN.O_Range_Warn" : Bool AT %DB5027.DBX48.7, 500 ms
   "2905RS001A01L01.trend_tag_name" : TextRef, internal   // Еденицы измерения При експорте из ECS через скрипт - заполняется автоматически, если теги копируются в ручную то требуется задатать свойство Text - имя тега для тренда
   "2905RS001A01L01.DQ.AL_H3" : Bool AT %DB5027.DBX16.0, 500 ms
   "2905RS001A01L01.DQ.AL_H2" : Bool AT %DB5027.DBX16.1, 500 ms
   "2905RS001A01L01.DQ.AL_H1" : Bool AT %DB5027.DBX16.2, 500 ms
   "2905RS001A01L01.DQ.AL_L1" : Bool AT %DB5027.DBX16.3, 500 ms
   "2905RS001A01L01.DQ.AL_L2" : Bool AT %DB5027.DBX16.4, 500 ms
   "2905RS001A01L01.DQ.AL_L3" : Bool AT %DB5027.DBX16.5, 500 ms
   "2905RS001A01L01.DQ.SIG_OK" : Bool AT %DB5027.DBX16.6, 500 ms
   "2905RS001A01L01.DQ.LIM_H2" : Bool AT %DB5027.DBX16.7, 500 ms
   "2905RS001A01L01.DQ.LIM_H1" : Bool AT %DB5027.DBX17.0, 500 ms
   "2905RS001A01L01.DQ.LIM_L1" : Bool AT %DB5027.DBX17.1, 500 ms
   "2905RS001A01L01.DQ.LIM_L2" : Bool AT %DB5027.DBX17.2, 500 ms
   "2905RS001A01L01.DQ.GR_P" : Bool AT %DB5027.DBX17.3, 500 ms
   "2905RS001A01L01.DQ.GR_N" : Bool AT %DB5027.DBX17.4, 500 ms
   "2905RS001A01L01.I.IN" : Real AT %DB5027.DBD2, 500 ms
   "2905RS001A01L01.I.SIG_TYPE" : Int AT %DB5027.DBW0, 500 ms
   "2905RS001A01L01.I.FI_BUS" : Byte AT %DB5027.DBB6, 500 ms
   "2905RS001A01L01.DI.U_RANGE" : Bool AT %DB5027.DBX7.0, 500 ms
   "2905RS001A01L01.DI.O_RANGE" : Bool AT %DB5027.DBX7.1, 500 ms
   "2905RS001A01L01.DI.SIG_FAULT" : Bool AT %DB5027.DBX7.2, 500 ms
   "2905RS001A01L01.DI.EnConfig" : Bool AT %DB5027.DBX7.3, 500 ms
   "2905RS001A01L01.DI.AEN" : Bool AT %DB5027.DBX7.4, 500 ms
   "2905RS001A01L01.DI.AL_SUPR" : Bool AT %DB5027.DBX7.5, 500 ms
   "2905RS001A01L01.Q.PV_NORM" : Real AT %DB5027.DBD8, 500 ms
   "2905RS001A01L01.Q.PV_SCAL" : Real AT %DB5027.DBD12, 500 ms
   "2905RS001A01L01.ParentInfo" : TextRef, internal   // Имя родителя для попап окна, вкладка инфо. При експорте из ECS через скрипт заполняется автоматически, если теги копируются в ручную то требуется в ручную задатать свойство Start Value

HMI tags "2910RS001A01F01"
   "2910RS001A01F01.MSW" : 52809b66-421d-457f-8884-6f7a49d4e247 AT %DB5030.DBX18.0, 500 ms
   "2910RS001A01F01.DefaultText" : TextRef, internal   // Заголовок POPUP окна. При експорте из ECS через скрипт заполняется автоматически, если теги копируются в ручную то требуется в ручную задатать свойство Start Value
   "2910RS001A01F01.BlockInfo" : Array [0..2] of Int AT %DB5030.DBX38.0, 500 ms
   "2910RS001A01F01.StatusWork" : Int AT %DB5030.DBW242, 500 ms
   "2910RS001A01F01.FP_PARAM.DampingTime" : Int AT %DB5030.DBW50, 500 ms
   "2910RS001A01F01.FP_PARAM.Force_Value" : Real AT %DB5030.DBD52, 500 ms
   "2910RS001A01F01.FP_PARAM.Scale_Min" : Real AT %DB5030.DBD56, 500 ms
   "2910RS001A01F01.FP_PARAM.Scale_Max" : Real AT %DB5030.DBD60, 500 ms
   "2910RS001A01F01.FP_PARAM.Gradient" : Real AT %DB5030.DBD64, 500 ms
   "2910RS001A01F01.FP_PARAM.Grad_Pos" : Real AT %DB5030.DBD68, 500 ms
   "2910RS001A01F01.FP_PARAM.Grad_Neg" : Real AT %DB5030.DBD72, 500 ms
   "2910RS001A01F01.FP_PARAM.Grad_X" : Real AT %DB5030.DBD76, 500 ms
   "2910RS001A01F01.FP_PARAM.Gradient_Time_Pre" : Int AT %DB5030.DBW80, 500 ms
   "2910RS001A01F01.FP_PARAM.Gradient_Time_ACC" : Int AT %DB5030.DBW82, 500 ms
   "2910RS001A01F01.FP_PARAM.Alarm_Hyst" : Real AT %DB5030.DBD84, 500 ms
   "2910RS001A01F01.FP_PARAM.AlarmLimit_H3" : Real AT %DB5030.DBD88, 500 ms
   "2910RS001A01F01.FP_PARAM.AlarmLimit_H2" : Real AT %DB5030.DBD92, 500 ms
   "2910RS001A01F01.FP_PARAM.AlarmLimit_H1" : Real AT %DB5030.DBD96, 500 ms
   "2910RS001A01F01.FP_PARAM.AlarmLimit_L1" : Real AT %DB5030.DBD100, 500 ms
   "2910RS001A01F01.FP_PARAM.AlarmLimit_L2" : Real AT %DB5030.DBD104, 500 ms
   "2910RS001A01F01.FP_PARAM.AlarmLimit_L3" : Real AT %DB5030.DBD108, 500 ms
   "2910RS001A01F01.FP_PARAM.AlarmDelay_H3_Pre" : Int AT %DB5030.DBW112, 500 ms
   "2910RS001A01F01.FP_PARAM.AlarmDelay_H3_Acc" : Int AT %DB5030.DBW114, 500 ms
   "2910RS001A01F01.FP_PARAM.AlarmDelay_H2_Pre" : Int AT %DB5030.DBW116, 500 ms
   "2910RS001A01F01.FP_PARAM.AlarmDelay_H2_Acc" : Int AT %DB5030.DBW118, 500 ms
   "2910RS001A01F01.FP_PARAM.AlarmDelay_H1_Pre" : Int AT %DB5030.DBW120, 500 ms
   "2910RS001A01F01.FP_PARAM.AlarmDelay_H1_Acc" : Int AT %DB5030.DBW122, 500 ms
   "2910RS001A01F01.FP_PARAM.AlarmDelay_L1_Pre" : Int AT %DB5030.DBW124, 500 ms
   "2910RS001A01F01.FP_PARAM.AlarmDelay_L1_Acc" : Int AT %DB5030.DBW126, 500 ms
   "2910RS001A01F01.FP_PARAM.AlarmDelay_L2_Pre" : Int AT %DB5030.DBW128, 500 ms
   "2910RS001A01F01.FP_PARAM.AlarmDelay_L2_Acc" : Int AT %DB5030.DBW130, 500 ms
   "2910RS001A01F01.FP_PARAM.AlarmDelay_L3_Pre" : Int AT %DB5030.DBW132, 500 ms
   "2910RS001A01F01.FP_PARAM.AlarmDelay_L3_Acc" : Int AT %DB5030.DBW134, 500 ms
   "2910RS001A01F01.FP_PARAM.OpenLoopDelay_Pre" : Int AT %DB5030.DBW136, 500 ms
   "2910RS001A01F01.FP_PARAM.OpenLoopDelay_Acc" : Int AT %DB5030.DBW138, 500 ms
   "2910RS001A01F01.FP_PARAM.OverRangeDelay_Pre" : Int AT %DB5030.DBW140, 500 ms
   "2910RS001A01F01.FP_PARAM.OverRangeDelay_Acc" : Int AT %DB5030.DBW142, 500 ms
   "2910RS001A01F01.FP_PARAM.AuxLimit_H2_Value" : Real AT %DB5030.DBD144, 500 ms
   "2910RS001A01F01.FP_PARAM.AuxLimit_H1_Value" : Real AT %DB5030.DBD148, 500 ms
   "2910RS001A01F01.FP_PARAM.AuxLimit_L2_Value" : Real AT %DB5030.DBD152, 500 ms
   "2910RS001A01F01.FP_PARAM.AuxLimit_L1_Value" : Real AT %DB5030.DBD156, 500 ms
   "2910RS001A01F01.Unit" : TextRef, internal   // Еденицы измерения При експорте из ECS через скрипт заполняется автоматически, если теги копируются в ручную то требуется задатать свойство Text
   "2910RS001A01F01.Decimals" : TextRef, internal   // Формат отображения При експорте из ECS через скрипт, заполняется автоматически. Если теги копируются в ручную то требуется задатать свойство Text s999999.9
   "2910RS001A01F01.FP_EN.Square" : Bool AT %DB5030.DBX46.0, 500 ms
   "2910RS001A01F01.FP_EN.SquareRoot" : Bool AT %DB5030.DBX46.1, 500 ms
   "2910RS001A01F01.FP_EN.ParentSupress" : Bool AT %DB5030.DBX46.2, 500 ms
   "2910RS001A01F01.FP_EN.ParentSupressUnit" : Bool AT %DB5030.DBX46.3, 500 ms
   "2910RS001A01F01.FP_EN.Force" : Bool AT %DB5030.DBX46.4, 500 ms
   "2910RS001A01F01.FP_EN.Damping" : Bool AT %DB5030.DBX46.5, 500 ms
   "2910RS001A01F01.FP_EN.Gradient_Pos" : Bool AT %DB5030.DBX46.6, 500 ms
   "2910RS001A01F01.FP_EN.Gradient_Neg" : Bool AT %DB5030.DBX46.7, 500 ms
   "2910RS001A01F01.FP_EN.Hysteresis" : Bool AT %DB5030.DBX47.0, 500 ms
   "2910RS001A01F01.FP_EN.Alarm_H3" : Bool AT %DB5030.DBX47.1, 500 ms
   "2910RS001A01F01.FP_EN.Alarm_H2" : Bool AT %DB5030.DBX47.2, 500 ms
   "2910RS001A01F01.FP_EN.Alarm_H1" : Bool AT %DB5030.DBX47.3, 500 ms
   "2910RS001A01F01.FP_EN.Alarm_L1" : Bool AT %DB5030.DBX47.4, 500 ms
   "2910RS001A01F01.FP_EN.Alarm_L2" : Bool AT %DB5030.DBX47.5, 500 ms
   "2910RS001A01F01.FP_EN.Alarm_L3" : Bool AT %DB5030.DBX47.6, 500 ms
   "2910RS001A01F01.FP_EN.AlarmDelay_H3" : Bool AT %DB5030.DBX47.7, 500 ms
   "2910RS001A01F01.FP_EN.AlarmDelay_H2" : Bool AT %DB5030.DBX48.0, 500 ms
   "2910RS001A01F01.FP_EN.AlarmDelay_H1" : Bool AT %DB5030.DBX48.1, 500 ms
   "2910RS001A01F01.FP_EN.AlarmDelay_L1" : Bool AT %DB5030.DBX48.2, 500 ms
   "2910RS001A01F01.FP_EN.AlarmDelay_L2" : Bool AT %DB5030.DBX48.3, 500 ms
   "2910RS001A01F01.FP_EN.AlarmDelay_L3" : Bool AT %DB5030.DBX48.4, 500 ms
   "2910RS001A01F01.FP_EN.ROC_Warn" : Bool AT %DB5030.DBX48.5, 500 ms
   "2910RS001A01F01.FP_EN.U_Range_Warn" : Bool AT %DB5030.DBX48.6, 500 ms
   "2910RS001A01F01.FP_EN.O_Range_Warn" : Bool AT %DB5030.DBX48.7, 500 ms
   "2910RS001A01F01.trend_tag_name" : TextRef, internal   // Еденицы измерения При експорте из ECS через скрипт - заполняется автоматически, если теги копируются в ручную то требуется задатать свойство Text - имя тега для тренда
   "2910RS001A01F01.DQ.AL_H3" : Bool AT %DB5030.DBX16.0, 500 ms
   "2910RS001A01F01.DQ.AL_H2" : Bool AT %DB5030.DBX16.1, 500 ms
   "2910RS001A01F01.DQ.AL_H1" : Bool AT %DB5030.DBX16.2, 500 ms
   "2910RS001A01F01.DQ.AL_L1" : Bool AT %DB5030.DBX16.3, 500 ms
   "2910RS001A01F01.DQ.AL_L2" : Bool AT %DB5030.DBX16.4, 500 ms
   "2910RS001A01F01.DQ.AL_L3" : Bool AT %DB5030.DBX16.5, 500 ms
   "2910RS001A01F01.DQ.SIG_OK" : Bool AT %DB5030.DBX16.6, 500 ms
   "2910RS001A01F01.DQ.LIM_H2" : Bool AT %DB5030.DBX16.7, 500 ms
   "2910RS001A01F01.DQ.LIM_H1" : Bool AT %DB5030.DBX17.0, 500 ms
   "2910RS001A01F01.DQ.LIM_L1" : Bool AT %DB5030.DBX17.1, 500 ms
   "2910RS001A01F01.DQ.LIM_L2" : Bool AT %DB5030.DBX17.2, 500 ms
   "2910RS001A01F01.DQ.GR_P" : Bool AT %DB5030.DBX17.3, 500 ms
   "2910RS001A01F01.DQ.GR_N" : Bool AT %DB5030.DBX17.4, 500 ms
   "2910RS001A01F01.I.IN" : Real AT %DB5030.DBD2, 500 ms
   "2910RS001A01F01.I.SIG_TYPE" : Int AT %DB5030.DBW0, 500 ms
   "2910RS001A01F01.I.FI_BUS" : Byte AT %DB5030.DBB6, 500 ms
   "2910RS001A01F01.DI.U_RANGE" : Bool AT %DB5030.DBX7.0, 500 ms
   "2910RS001A01F01.DI.O_RANGE" : Bool AT %DB5030.DBX7.1, 500 ms
   "2910RS001A01F01.DI.SIG_FAULT" : Bool AT %DB5030.DBX7.2, 500 ms
   "2910RS001A01F01.DI.EnConfig" : Bool AT %DB5030.DBX7.3, 500 ms
   "2910RS001A01F01.DI.AEN" : Bool AT %DB5030.DBX7.4, 500 ms
   "2910RS001A01F01.DI.AL_SUPR" : Bool AT %DB5030.DBX7.5, 500 ms
   "2910RS001A01F01.Q.PV_NORM" : Real AT %DB5030.DBD8, 500 ms
   "2910RS001A01F01.Q.PV_SCAL" : Real AT %DB5030.DBD12, 500 ms
   "2910RS001A01F01.ParentInfo" : TextRef, internal   // Имя родителя для попап окна, вкладка инфо. При експорте из ECS через скрипт заполняется автоматически, если теги копируются в ручную то требуется в ручную задатать свойство Start Value

HMI tags "2910RS001A01L01"
   "2910RS001A01L01.MSW" : 52809b66-421d-457f-8884-6f7a49d4e247 AT %DB5031.DBX18.0, 500 ms
   "2910RS001A01L01.DefaultText" : TextRef, internal   // Заголовок POPUP окна. При експорте из ECS через скрипт заполняется автоматически, если теги копируются в ручную то требуется в ручную задатать свойство Start Value
   "2910RS001A01L01.BlockInfo" : Array [0..2] of Int AT %DB5031.DBX38.0, 500 ms
   "2910RS001A01L01.StatusWork" : Int AT %DB5031.DBW242, 500 ms
   "2910RS001A01L01.FP_PARAM.DampingTime" : Int AT %DB5031.DBW50, 500 ms
   "2910RS001A01L01.FP_PARAM.Force_Value" : Real AT %DB5031.DBD52, 500 ms
   "2910RS001A01L01.FP_PARAM.Scale_Min" : Real AT %DB5031.DBD56, 500 ms
   "2910RS001A01L01.FP_PARAM.Scale_Max" : Real AT %DB5031.DBD60, 500 ms
   "2910RS001A01L01.FP_PARAM.Gradient" : Real AT %DB5031.DBD64, 500 ms
   "2910RS001A01L01.FP_PARAM.Grad_Pos" : Real AT %DB5031.DBD68, 500 ms
   "2910RS001A01L01.FP_PARAM.Grad_Neg" : Real AT %DB5031.DBD72, 500 ms
   "2910RS001A01L01.FP_PARAM.Grad_X" : Real AT %DB5031.DBD76, 500 ms
   "2910RS001A01L01.FP_PARAM.Gradient_Time_Pre" : Int AT %DB5031.DBW80, 500 ms
   "2910RS001A01L01.FP_PARAM.Gradient_Time_ACC" : Int AT %DB5031.DBW82, 500 ms
   "2910RS001A01L01.FP_PARAM.Alarm_Hyst" : Real AT %DB5031.DBD84, 500 ms
   "2910RS001A01L01.FP_PARAM.AlarmLimit_H3" : Real AT %DB5031.DBD88, 500 ms
   "2910RS001A01L01.FP_PARAM.AlarmLimit_H2" : Real AT %DB5031.DBD92, 500 ms
   "2910RS001A01L01.FP_PARAM.AlarmLimit_H1" : Real AT %DB5031.DBD96, 500 ms
   "2910RS001A01L01.FP_PARAM.AlarmLimit_L1" : Real AT %DB5031.DBD100, 500 ms
   "2910RS001A01L01.FP_PARAM.AlarmLimit_L2" : Real AT %DB5031.DBD104, 500 ms
   "2910RS001A01L01.FP_PARAM.AlarmLimit_L3" : Real AT %DB5031.DBD108, 500 ms
   "2910RS001A01L01.FP_PARAM.AlarmDelay_H3_Pre" : Int AT %DB5031.DBW112, 500 ms
   "2910RS001A01L01.FP_PARAM.AlarmDelay_H3_Acc" : Int AT %DB5031.DBW114, 500 ms
   "2910RS001A01L01.FP_PARAM.AlarmDelay_H2_Pre" : Int AT %DB5031.DBW116, 500 ms
   "2910RS001A01L01.FP_PARAM.AlarmDelay_H2_Acc" : Int AT %DB5031.DBW118, 500 ms
   "2910RS001A01L01.FP_PARAM.AlarmDelay_H1_Pre" : Int AT %DB5031.DBW120, 500 ms
   "2910RS001A01L01.FP_PARAM.AlarmDelay_H1_Acc" : Int AT %DB5031.DBW122, 500 ms
   "2910RS001A01L01.FP_PARAM.AlarmDelay_L1_Pre" : Int AT %DB5031.DBW124, 500 ms
   "2910RS001A01L01.FP_PARAM.AlarmDelay_L1_Acc" : Int AT %DB5031.DBW126, 500 ms
   "2910RS001A01L01.FP_PARAM.AlarmDelay_L2_Pre" : Int AT %DB5031.DBW128, 500 ms
   "2910RS001A01L01.FP_PARAM.AlarmDelay_L2_Acc" : Int AT %DB5031.DBW130, 500 ms
   "2910RS001A01L01.FP_PARAM.AlarmDelay_L3_Pre" : Int AT %DB5031.DBW132, 500 ms
   "2910RS001A01L01.FP_PARAM.AlarmDelay_L3_Acc" : Int AT %DB5031.DBW134, 500 ms
   "2910RS001A01L01.FP_PARAM.OpenLoopDelay_Pre" : Int AT %DB5031.DBW136, 500 ms
   "2910RS001A01L01.FP_PARAM.OpenLoopDelay_Acc" : Int AT %DB5031.DBW138, 500 ms
   "2910RS001A01L01.FP_PARAM.OverRangeDelay_Pre" : Int AT %DB5031.DBW140, 500 ms
   "2910RS001A01L01.FP_PARAM.OverRangeDelay_Acc" : Int AT %DB5031.DBW142, 500 ms
   "2910RS001A01L01.FP_PARAM.AuxLimit_H2_Value" : Real AT %DB5031.DBD144, 500 ms
   "2910RS001A01L01.FP_PARAM.AuxLimit_H1_Value" : Real AT %DB5031.DBD148, 500 ms
   "2910RS001A01L01.FP_PARAM.AuxLimit_L2_Value" : Real AT %DB5031.DBD152, 500 ms
   "2910RS001A01L01.FP_PARAM.AuxLimit_L1_Value" : Real AT %DB5031.DBD156, 500 ms
   "2910RS001A01L01.Unit" : TextRef, internal   // Еденицы измерения При експорте из ECS через скрипт заполняется автоматически, если теги копируются в ручную то требуется задатать свойство Text
   "2910RS001A01L01.Decimals" : TextRef, internal   // Формат отображения При експорте из ECS через скрипт, заполняется автоматически. Если теги копируются в ручную то требуется задатать свойство Text s999999.9
   "2910RS001A01L01.FP_EN.Square" : Bool AT %DB5031.DBX46.0, 500 ms
   "2910RS001A01L01.FP_EN.SquareRoot" : Bool AT %DB5031.DBX46.1, 500 ms
   "2910RS001A01L01.FP_EN.ParentSupress" : Bool AT %DB5031.DBX46.2, 500 ms
   "2910RS001A01L01.FP_EN.ParentSupressUnit" : Bool AT %DB5031.DBX46.3, 500 ms
   "2910RS001A01L01.FP_EN.Force" : Bool AT %DB5031.DBX46.4, 500 ms
   "2910RS001A01L01.FP_EN.Damping" : Bool AT %DB5031.DBX46.5, 500 ms
   "2910RS001A01L01.FP_EN.Gradient_Pos" : Bool AT %DB5031.DBX46.6, 500 ms
   "2910RS001A01L01.FP_EN.Gradient_Neg" : Bool AT %DB5031.DBX46.7, 500 ms
   "2910RS001A01L01.FP_EN.Hysteresis" : Bool AT %DB5031.DBX47.0, 500 ms
   "2910RS001A01L01.FP_EN.Alarm_H3" : Bool AT %DB5031.DBX47.1, 500 ms
   "2910RS001A01L01.FP_EN.Alarm_H2" : Bool AT %DB5031.DBX47.2, 500 ms
   "2910RS001A01L01.FP_EN.Alarm_H1" : Bool AT %DB5031.DBX47.3, 500 ms
   "2910RS001A01L01.FP_EN.Alarm_L1" : Bool AT %DB5031.DBX47.4, 500 ms
   "2910RS001A01L01.FP_EN.Alarm_L2" : Bool AT %DB5031.DBX47.5, 500 ms
   "2910RS001A01L01.FP_EN.Alarm_L3" : Bool AT %DB5031.DBX47.6, 500 ms
   "2910RS001A01L01.FP_EN.AlarmDelay_H3" : Bool AT %DB5031.DBX47.7, 500 ms
   "2910RS001A01L01.FP_EN.AlarmDelay_H2" : Bool AT %DB5031.DBX48.0, 500 ms
   "2910RS001A01L01.FP_EN.AlarmDelay_H1" : Bool AT %DB5031.DBX48.1, 500 ms
   "2910RS001A01L01.FP_EN.AlarmDelay_L1" : Bool AT %DB5031.DBX48.2, 500 ms
   "2910RS001A01L01.FP_EN.AlarmDelay_L2" : Bool AT %DB5031.DBX48.3, 500 ms
   "2910RS001A01L01.FP_EN.AlarmDelay_L3" : Bool AT %DB5031.DBX48.4, 500 ms
   "2910RS001A01L01.FP_EN.ROC_Warn" : Bool AT %DB5031.DBX48.5, 500 ms
   "2910RS001A01L01.FP_EN.U_Range_Warn" : Bool AT %DB5031.DBX48.6, 500 ms
   "2910RS001A01L01.FP_EN.O_Range_Warn" : Bool AT %DB5031.DBX48.7, 500 ms
   "2910RS001A01L01.trend_tag_name" : TextRef, internal   // Еденицы измерения При експорте из ECS через скрипт - заполняется автоматически, если теги копируются в ручную то требуется задатать свойство Text - имя тега для тренда
   "2910RS001A01L01.DQ.AL_H3" : Bool AT %DB5031.DBX16.0, 500 ms
   "2910RS001A01L01.DQ.AL_H2" : Bool AT %DB5031.DBX16.1, 500 ms
   "2910RS001A01L01.DQ.AL_H1" : Bool AT %DB5031.DBX16.2, 500 ms
   "2910RS001A01L01.DQ.AL_L1" : Bool AT %DB5031.DBX16.3, 500 ms
   "2910RS001A01L01.DQ.AL_L2" : Bool AT %DB5031.DBX16.4, 500 ms
   "2910RS001A01L01.DQ.AL_L3" : Bool AT %DB5031.DBX16.5, 500 ms
   "2910RS001A01L01.DQ.SIG_OK" : Bool AT %DB5031.DBX16.6, 500 ms
   "2910RS001A01L01.DQ.LIM_H2" : Bool AT %DB5031.DBX16.7, 500 ms
   "2910RS001A01L01.DQ.LIM_H1" : Bool AT %DB5031.DBX17.0, 500 ms
   "2910RS001A01L01.DQ.LIM_L1" : Bool AT %DB5031.DBX17.1, 500 ms
   "2910RS001A01L01.DQ.LIM_L2" : Bool AT %DB5031.DBX17.2, 500 ms
   "2910RS001A01L01.DQ.GR_P" : Bool AT %DB5031.DBX17.3, 500 ms
   "2910RS001A01L01.DQ.GR_N" : Bool AT %DB5031.DBX17.4, 500 ms
   "2910RS001A01L01.I.IN" : Real AT %DB5031.DBD2, 500 ms
   "2910RS001A01L01.I.SIG_TYPE" : Int AT %DB5031.DBW0, 500 ms
   "2910RS001A01L01.I.FI_BUS" : Byte AT %DB5031.DBB6, 500 ms
   "2910RS001A01L01.DI.U_RANGE" : Bool AT %DB5031.DBX7.0, 500 ms
   "2910RS001A01L01.DI.O_RANGE" : Bool AT %DB5031.DBX7.1, 500 ms
   "2910RS001A01L01.DI.SIG_FAULT" : Bool AT %DB5031.DBX7.2, 500 ms
   "2910RS001A01L01.DI.EnConfig" : Bool AT %DB5031.DBX7.3, 500 ms
   "2910RS001A01L01.DI.AEN" : Bool AT %DB5031.DBX7.4, 500 ms
   "2910RS001A01L01.DI.AL_SUPR" : Bool AT %DB5031.DBX7.5, 500 ms
   "2910RS001A01L01.Q.PV_NORM" : Real AT %DB5031.DBD8, 500 ms
   "2910RS001A01L01.Q.PV_SCAL" : Real AT %DB5031.DBD12, 500 ms
   "2910RS001A01L01.ParentInfo" : TextRef, internal   // Имя родителя для попап окна, вкладка инфо. При експорте из ECS через скрипт заполняется автоматически, если теги копируются в ручную то требуется в ручную задатать свойство Start Value

HMI tags "2910RS001A01L02"
   "2910RS001A01L02.MSW" : 52809b66-421d-457f-8884-6f7a49d4e247 AT %DB5032.DBX18.0, 500 ms
   "2910RS001A01L02.DefaultText" : TextRef, internal   // Заголовок POPUP окна. При експорте из ECS через скрипт заполняется автоматически, если теги копируются в ручную то требуется в ручную задатать свойство Start Value
   "2910RS001A01L02.BlockInfo" : Array [0..2] of Int AT %DB5032.DBX38.0, 500 ms
   "2910RS001A01L02.StatusWork" : Int AT %DB5032.DBW242, 500 ms
   "2910RS001A01L02.FP_PARAM.DampingTime" : Int AT %DB5032.DBW50, 500 ms
   "2910RS001A01L02.FP_PARAM.Force_Value" : Real AT %DB5032.DBD52, 500 ms
   "2910RS001A01L02.FP_PARAM.Scale_Min" : Real AT %DB5032.DBD56, 500 ms
   "2910RS001A01L02.FP_PARAM.Scale_Max" : Real AT %DB5032.DBD60, 500 ms
   "2910RS001A01L02.FP_PARAM.Gradient" : Real AT %DB5032.DBD64, 500 ms
   "2910RS001A01L02.FP_PARAM.Grad_Pos" : Real AT %DB5032.DBD68, 500 ms
   "2910RS001A01L02.FP_PARAM.Grad_Neg" : Real AT %DB5032.DBD72, 500 ms
   "2910RS001A01L02.FP_PARAM.Grad_X" : Real AT %DB5032.DBD76, 500 ms
   "2910RS001A01L02.FP_PARAM.Gradient_Time_Pre" : Int AT %DB5032.DBW80, 500 ms
   "2910RS001A01L02.FP_PARAM.Gradient_Time_ACC" : Int AT %DB5032.DBW82, 500 ms
   "2910RS001A01L02.FP_PARAM.Alarm_Hyst" : Real AT %DB5032.DBD84, 500 ms
   "2910RS001A01L02.FP_PARAM.AlarmLimit_H3" : Real AT %DB5032.DBD88, 500 ms
   "2910RS001A01L02.FP_PARAM.AlarmLimit_H2" : Real AT %DB5032.DBD92, 500 ms
   "2910RS001A01L02.FP_PARAM.AlarmLimit_H1" : Real AT %DB5032.DBD96, 500 ms
   "2910RS001A01L02.FP_PARAM.AlarmLimit_L1" : Real AT %DB5032.DBD100, 500 ms
   "2910RS001A01L02.FP_PARAM.AlarmLimit_L2" : Real AT %DB5032.DBD104, 500 ms
   "2910RS001A01L02.FP_PARAM.AlarmLimit_L3" : Real AT %DB5032.DBD108, 500 ms
   "2910RS001A01L02.FP_PARAM.AlarmDelay_H3_Pre" : Int AT %DB5032.DBW112, 500 ms
   "2910RS001A01L02.FP_PARAM.AlarmDelay_H3_Acc" : Int AT %DB5032.DBW114, 500 ms
   "2910RS001A01L02.FP_PARAM.AlarmDelay_H2_Pre" : Int AT %DB5032.DBW116, 500 ms
   "2910RS001A01L02.FP_PARAM.AlarmDelay_H2_Acc" : Int AT %DB5032.DBW118, 500 ms
   "2910RS001A01L02.FP_PARAM.AlarmDelay_H1_Pre" : Int AT %DB5032.DBW120, 500 ms
   "2910RS001A01L02.FP_PARAM.AlarmDelay_H1_Acc" : Int AT %DB5032.DBW122, 500 ms
   "2910RS001A01L02.FP_PARAM.AlarmDelay_L1_Pre" : Int AT %DB5032.DBW124, 500 ms
   "2910RS001A01L02.FP_PARAM.AlarmDelay_L1_Acc" : Int AT %DB5032.DBW126, 500 ms
   "2910RS001A01L02.FP_PARAM.AlarmDelay_L2_Pre" : Int AT %DB5032.DBW128, 500 ms
   "2910RS001A01L02.FP_PARAM.AlarmDelay_L2_Acc" : Int AT %DB5032.DBW130, 500 ms
   "2910RS001A01L02.FP_PARAM.AlarmDelay_L3_Pre" : Int AT %DB5032.DBW132, 500 ms
   "2910RS001A01L02.FP_PARAM.AlarmDelay_L3_Acc" : Int AT %DB5032.DBW134, 500 ms
   "2910RS001A01L02.FP_PARAM.OpenLoopDelay_Pre" : Int AT %DB5032.DBW136, 500 ms
   "2910RS001A01L02.FP_PARAM.OpenLoopDelay_Acc" : Int AT %DB5032.DBW138, 500 ms
   "2910RS001A01L02.FP_PARAM.OverRangeDelay_Pre" : Int AT %DB5032.DBW140, 500 ms
   "2910RS001A01L02.FP_PARAM.OverRangeDelay_Acc" : Int AT %DB5032.DBW142, 500 ms
   "2910RS001A01L02.FP_PARAM.AuxLimit_H2_Value" : Real AT %DB5032.DBD144, 500 ms
   "2910RS001A01L02.FP_PARAM.AuxLimit_H1_Value" : Real AT %DB5032.DBD148, 500 ms
   "2910RS001A01L02.FP_PARAM.AuxLimit_L2_Value" : Real AT %DB5032.DBD152, 500 ms
   "2910RS001A01L02.FP_PARAM.AuxLimit_L1_Value" : Real AT %DB5032.DBD156, 500 ms
   "2910RS001A01L02.Unit" : TextRef, internal   // Еденицы измерения При експорте из ECS через скрипт заполняется автоматически, если теги копируются в ручную то требуется задатать свойство Text
   "2910RS001A01L02.Decimals" : TextRef, internal   // Формат отображения При експорте из ECS через скрипт, заполняется автоматически. Если теги копируются в ручную то требуется задатать свойство Text s999999.9
   "2910RS001A01L02.FP_EN.Square" : Bool AT %DB5032.DBX46.0, 500 ms
   "2910RS001A01L02.FP_EN.SquareRoot" : Bool AT %DB5032.DBX46.1, 500 ms
   "2910RS001A01L02.FP_EN.ParentSupress" : Bool AT %DB5032.DBX46.2, 500 ms
   "2910RS001A01L02.FP_EN.ParentSupressUnit" : Bool AT %DB5032.DBX46.3, 500 ms
   "2910RS001A01L02.FP_EN.Force" : Bool AT %DB5032.DBX46.4, 500 ms
   "2910RS001A01L02.FP_EN.Damping" : Bool AT %DB5032.DBX46.5, 500 ms
   "2910RS001A01L02.FP_EN.Gradient_Pos" : Bool AT %DB5032.DBX46.6, 500 ms
   "2910RS001A01L02.FP_EN.Gradient_Neg" : Bool AT %DB5032.DBX46.7, 500 ms
   "2910RS001A01L02.FP_EN.Hysteresis" : Bool AT %DB5032.DBX47.0, 500 ms
   "2910RS001A01L02.FP_EN.Alarm_H3" : Bool AT %DB5032.DBX47.1, 500 ms
   "2910RS001A01L02.FP_EN.Alarm_H2" : Bool AT %DB5032.DBX47.2, 500 ms
   "2910RS001A01L02.FP_EN.Alarm_H1" : Bool AT %DB5032.DBX47.3, 500 ms
   "2910RS001A01L02.FP_EN.Alarm_L1" : Bool AT %DB5032.DBX47.4, 500 ms
   "2910RS001A01L02.FP_EN.Alarm_L2" : Bool AT %DB5032.DBX47.5, 500 ms
   "2910RS001A01L02.FP_EN.Alarm_L3" : Bool AT %DB5032.DBX47.6, 500 ms
   "2910RS001A01L02.FP_EN.AlarmDelay_H3" : Bool AT %DB5032.DBX47.7, 500 ms
   "2910RS001A01L02.FP_EN.AlarmDelay_H2" : Bool AT %DB5032.DBX48.0, 500 ms
   "2910RS001A01L02.FP_EN.AlarmDelay_H1" : Bool AT %DB5032.DBX48.1, 500 ms
   "2910RS001A01L02.FP_EN.AlarmDelay_L1" : Bool AT %DB5032.DBX48.2, 500 ms
   "2910RS001A01L02.FP_EN.AlarmDelay_L2" : Bool AT %DB5032.DBX48.3, 500 ms
   "2910RS001A01L02.FP_EN.AlarmDelay_L3" : Bool AT %DB5032.DBX48.4, 500 ms
   "2910RS001A01L02.FP_EN.ROC_Warn" : Bool AT %DB5032.DBX48.5, 500 ms
   "2910RS001A01L02.FP_EN.U_Range_Warn" : Bool AT %DB5032.DBX48.6, 500 ms
   "2910RS001A01L02.FP_EN.O_Range_Warn" : Bool AT %DB5032.DBX48.7, 500 ms
   "2910RS001A01L02.trend_tag_name" : TextRef, internal   // Еденицы измерения При експорте из ECS через скрипт - заполняется автоматически, если теги копируются в ручную то требуется задатать свойство Text - имя тега для тренда
   "2910RS001A01L02.DQ.AL_H3" : Bool AT %DB5032.DBX16.0, 500 ms
   "2910RS001A01L02.DQ.AL_H2" : Bool AT %DB5032.DBX16.1, 500 ms
   "2910RS001A01L02.DQ.AL_H1" : Bool AT %DB5032.DBX16.2, 500 ms
   "2910RS001A01L02.DQ.AL_L1" : Bool AT %DB5032.DBX16.3, 500 ms
   "2910RS001A01L02.DQ.AL_L2" : Bool AT %DB5032.DBX16.4, 500 ms
   "2910RS001A01L02.DQ.AL_L3" : Bool AT %DB5032.DBX16.5, 500 ms
   "2910RS001A01L02.DQ.SIG_OK" : Bool AT %DB5032.DBX16.6, 500 ms
   "2910RS001A01L02.DQ.LIM_H2" : Bool AT %DB5032.DBX16.7, 500 ms
   "2910RS001A01L02.DQ.LIM_H1" : Bool AT %DB5032.DBX17.0, 500 ms
   "2910RS001A01L02.DQ.LIM_L1" : Bool AT %DB5032.DBX17.1, 500 ms
   "2910RS001A01L02.DQ.LIM_L2" : Bool AT %DB5032.DBX17.2, 500 ms
   "2910RS001A01L02.DQ.GR_P" : Bool AT %DB5032.DBX17.3, 500 ms
   "2910RS001A01L02.DQ.GR_N" : Bool AT %DB5032.DBX17.4, 500 ms
   "2910RS001A01L02.I.IN" : Real AT %DB5032.DBD2, 500 ms
   "2910RS001A01L02.I.SIG_TYPE" : Int AT %DB5032.DBW0, 500 ms
   "2910RS001A01L02.I.FI_BUS" : Byte AT %DB5032.DBB6, 500 ms
   "2910RS001A01L02.DI.U_RANGE" : Bool AT %DB5032.DBX7.0, 500 ms
   "2910RS001A01L02.DI.O_RANGE" : Bool AT %DB5032.DBX7.1, 500 ms
   "2910RS001A01L02.DI.SIG_FAULT" : Bool AT %DB5032.DBX7.2, 500 ms
   "2910RS001A01L02.DI.EnConfig" : Bool AT %DB5032.DBX7.3, 500 ms
   "2910RS001A01L02.DI.AEN" : Bool AT %DB5032.DBX7.4, 500 ms
   "2910RS001A01L02.DI.AL_SUPR" : Bool AT %DB5032.DBX7.5, 500 ms
   "2910RS001A01L02.Q.PV_NORM" : Real AT %DB5032.DBD8, 500 ms
   "2910RS001A01L02.Q.PV_SCAL" : Real AT %DB5032.DBD12, 500 ms
   "2910RS001A01L02.ParentInfo" : TextRef, internal   // Имя родителя для попап окна, вкладка инфо. При експорте из ECS через скрипт заполняется автоматически, если теги копируются в ручную то требуется в ручную задатать свойство Start Value

HMI tags "2910RS001A01N01"
   "2910RS001A01N01.MSW" : 52809b66-421d-457f-8884-6f7a49d4e247 AT %DB5033.DBX18.0, 500 ms
   "2910RS001A01N01.DefaultText" : TextRef, internal   // Заголовок POPUP окна. При експорте из ECS через скрипт заполняется автоматически, если теги копируются в ручную то требуется в ручную задатать свойство Start Value
   "2910RS001A01N01.BlockInfo" : Array [0..2] of Int AT %DB5033.DBX38.0, 500 ms
   "2910RS001A01N01.StatusWork" : Int AT %DB5033.DBW242, 500 ms
   "2910RS001A01N01.FP_PARAM.DampingTime" : Int AT %DB5033.DBW50, 500 ms
   "2910RS001A01N01.FP_PARAM.Force_Value" : Real AT %DB5033.DBD52, 500 ms
   "2910RS001A01N01.FP_PARAM.Scale_Min" : Real AT %DB5033.DBD56, 500 ms
   "2910RS001A01N01.FP_PARAM.Scale_Max" : Real AT %DB5033.DBD60, 500 ms
   "2910RS001A01N01.FP_PARAM.Gradient" : Real AT %DB5033.DBD64, 500 ms
   "2910RS001A01N01.FP_PARAM.Grad_Pos" : Real AT %DB5033.DBD68, 500 ms
   "2910RS001A01N01.FP_PARAM.Grad_Neg" : Real AT %DB5033.DBD72, 500 ms
   "2910RS001A01N01.FP_PARAM.Grad_X" : Real AT %DB5033.DBD76, 500 ms
   "2910RS001A01N01.FP_PARAM.Gradient_Time_Pre" : Int AT %DB5033.DBW80, 500 ms
   "2910RS001A01N01.FP_PARAM.Gradient_Time_ACC" : Int AT %DB5033.DBW82, 500 ms
   "2910RS001A01N01.FP_PARAM.Alarm_Hyst" : Real AT %DB5033.DBD84, 500 ms
   "2910RS001A01N01.FP_PARAM.AlarmLimit_H3" : Real AT %DB5033.DBD88, 500 ms
   "2910RS001A01N01.FP_PARAM.AlarmLimit_H2" : Real AT %DB5033.DBD92, 500 ms
   "2910RS001A01N01.FP_PARAM.AlarmLimit_H1" : Real AT %DB5033.DBD96, 500 ms
   "2910RS001A01N01.FP_PARAM.AlarmLimit_L1" : Real AT %DB5033.DBD100, 500 ms
   "2910RS001A01N01.FP_PARAM.AlarmLimit_L2" : Real AT %DB5033.DBD104, 500 ms
   "2910RS001A01N01.FP_PARAM.AlarmLimit_L3" : Real AT %DB5033.DBD108, 500 ms
   "2910RS001A01N01.FP_PARAM.AlarmDelay_H3_Pre" : Int AT %DB5033.DBW112, 500 ms
   "2910RS001A01N01.FP_PARAM.AlarmDelay_H3_Acc" : Int AT %DB5033.DBW114, 500 ms
   "2910RS001A01N01.FP_PARAM.AlarmDelay_H2_Pre" : Int AT %DB5033.DBW116, 500 ms
   "2910RS001A01N01.FP_PARAM.AlarmDelay_H2_Acc" : Int AT %DB5033.DBW118, 500 ms
   "2910RS001A01N01.FP_PARAM.AlarmDelay_H1_Pre" : Int AT %DB5033.DBW120, 500 ms
   "2910RS001A01N01.FP_PARAM.AlarmDelay_H1_Acc" : Int AT %DB5033.DBW122, 500 ms
   "2910RS001A01N01.FP_PARAM.AlarmDelay_L1_Pre" : Int AT %DB5033.DBW124, 500 ms
   "2910RS001A01N01.FP_PARAM.AlarmDelay_L1_Acc" : Int AT %DB5033.DBW126, 500 ms
   "2910RS001A01N01.FP_PARAM.AlarmDelay_L2_Pre" : Int AT %DB5033.DBW128, 500 ms
   "2910RS001A01N01.FP_PARAM.AlarmDelay_L2_Acc" : Int AT %DB5033.DBW130, 500 ms
   "2910RS001A01N01.FP_PARAM.AlarmDelay_L3_Pre" : Int AT %DB5033.DBW132, 500 ms
   "2910RS001A01N01.FP_PARAM.AlarmDelay_L3_Acc" : Int AT %DB5033.DBW134, 500 ms
   "2910RS001A01N01.FP_PARAM.OpenLoopDelay_Pre" : Int AT %DB5033.DBW136, 500 ms
   "2910RS001A01N01.FP_PARAM.OpenLoopDelay_Acc" : Int AT %DB5033.DBW138, 500 ms
   "2910RS001A01N01.FP_PARAM.OverRangeDelay_Pre" : Int AT %DB5033.DBW140, 500 ms
   "2910RS001A01N01.FP_PARAM.OverRangeDelay_Acc" : Int AT %DB5033.DBW142, 500 ms
   "2910RS001A01N01.FP_PARAM.AuxLimit_H2_Value" : Real AT %DB5033.DBD144, 500 ms
   "2910RS001A01N01.FP_PARAM.AuxLimit_H1_Value" : Real AT %DB5033.DBD148, 500 ms
   "2910RS001A01N01.FP_PARAM.AuxLimit_L2_Value" : Real AT %DB5033.DBD152, 500 ms
   "2910RS001A01N01.FP_PARAM.AuxLimit_L1_Value" : Real AT %DB5033.DBD156, 500 ms
   "2910RS001A01N01.Unit" : TextRef, internal   // Еденицы измерения При експорте из ECS через скрипт заполняется автоматически, если теги копируются в ручную то требуется задатать свойство Text
   "2910RS001A01N01.Decimals" : TextRef, internal   // Формат отображения При експорте из ECS через скрипт, заполняется автоматически. Если теги копируются в ручную то требуется задатать свойство Text s999999.9
   "2910RS001A01N01.FP_EN.Square" : Bool AT %DB5033.DBX46.0, 500 ms
   "2910RS001A01N01.FP_EN.SquareRoot" : Bool AT %DB5033.DBX46.1, 500 ms
   "2910RS001A01N01.FP_EN.ParentSupress" : Bool AT %DB5033.DBX46.2, 500 ms
   "2910RS001A01N01.FP_EN.ParentSupressUnit" : Bool AT %DB5033.DBX46.3, 500 ms
   "2910RS001A01N01.FP_EN.Force" : Bool AT %DB5033.DBX46.4, 500 ms
   "2910RS001A01N01.FP_EN.Damping" : Bool AT %DB5033.DBX46.5, 500 ms
   "2910RS001A01N01.FP_EN.Gradient_Pos" : Bool AT %DB5033.DBX46.6, 500 ms
   "2910RS001A01N01.FP_EN.Gradient_Neg" : Bool AT %DB5033.DBX46.7, 500 ms
   "2910RS001A01N01.FP_EN.Hysteresis" : Bool AT %DB5033.DBX47.0, 500 ms
   "2910RS001A01N01.FP_EN.Alarm_H3" : Bool AT %DB5033.DBX47.1, 500 ms
   "2910RS001A01N01.FP_EN.Alarm_H2" : Bool AT %DB5033.DBX47.2, 500 ms
   "2910RS001A01N01.FP_EN.Alarm_H1" : Bool AT %DB5033.DBX47.3, 500 ms
   "2910RS001A01N01.FP_EN.Alarm_L1" : Bool AT %DB5033.DBX47.4, 500 ms
   "2910RS001A01N01.FP_EN.Alarm_L2" : Bool AT %DB5033.DBX47.5, 500 ms
   "2910RS001A01N01.FP_EN.Alarm_L3" : Bool AT %DB5033.DBX47.6, 500 ms
   "2910RS001A01N01.FP_EN.AlarmDelay_H3" : Bool AT %DB5033.DBX47.7, 500 ms
   "2910RS001A01N01.FP_EN.AlarmDelay_H2" : Bool AT %DB5033.DBX48.0, 500 ms
   "2910RS001A01N01.FP_EN.AlarmDelay_H1" : Bool AT %DB5033.DBX48.1, 500 ms
   "2910RS001A01N01.FP_EN.AlarmDelay_L1" : Bool AT %DB5033.DBX48.2, 500 ms
   "2910RS001A01N01.FP_EN.AlarmDelay_L2" : Bool AT %DB5033.DBX48.3, 500 ms
   "2910RS001A01N01.FP_EN.AlarmDelay_L3" : Bool AT %DB5033.DBX48.4, 500 ms
   "2910RS001A01N01.FP_EN.ROC_Warn" : Bool AT %DB5033.DBX48.5, 500 ms
   "2910RS001A01N01.FP_EN.U_Range_Warn" : Bool AT %DB5033.DBX48.6, 500 ms
   "2910RS001A01N01.FP_EN.O_Range_Warn" : Bool AT %DB5033.DBX48.7, 500 ms
   "2910RS001A01N01.trend_tag_name" : TextRef, internal   // Еденицы измерения При експорте из ECS через скрипт - заполняется автоматически, если теги копируются в ручную то требуется задатать свойство Text - имя тега для тренда
   "2910RS001A01N01.DQ.AL_H3" : Bool AT %DB5033.DBX16.0, 500 ms
   "2910RS001A01N01.DQ.AL_H2" : Bool AT %DB5033.DBX16.1, 500 ms
   "2910RS001A01N01.DQ.AL_H1" : Bool AT %DB5033.DBX16.2, 500 ms
   "2910RS001A01N01.DQ.AL_L1" : Bool AT %DB5033.DBX16.3, 500 ms
   "2910RS001A01N01.DQ.AL_L2" : Bool AT %DB5033.DBX16.4, 500 ms
   "2910RS001A01N01.DQ.AL_L3" : Bool AT %DB5033.DBX16.5, 500 ms
   "2910RS001A01N01.DQ.SIG_OK" : Bool AT %DB5033.DBX16.6, 500 ms
   "2910RS001A01N01.DQ.LIM_H2" : Bool AT %DB5033.DBX16.7, 500 ms
   "2910RS001A01N01.DQ.LIM_H1" : Bool AT %DB5033.DBX17.0, 500 ms
   "2910RS001A01N01.DQ.LIM_L1" : Bool AT %DB5033.DBX17.1, 500 ms
   "2910RS001A01N01.DQ.LIM_L2" : Bool AT %DB5033.DBX17.2, 500 ms
   "2910RS001A01N01.DQ.GR_P" : Bool AT %DB5033.DBX17.3, 500 ms
   "2910RS001A01N01.DQ.GR_N" : Bool AT %DB5033.DBX17.4, 500 ms
   "2910RS001A01N01.I.IN" : Real AT %DB5033.DBD2, 500 ms
   "2910RS001A01N01.I.SIG_TYPE" : Int AT %DB5033.DBW0, 500 ms
   "2910RS001A01N01.I.FI_BUS" : Byte AT %DB5033.DBB6, 500 ms
   "2910RS001A01N01.DI.U_RANGE" : Bool AT %DB5033.DBX7.0, 500 ms
   "2910RS001A01N01.DI.O_RANGE" : Bool AT %DB5033.DBX7.1, 500 ms
   "2910RS001A01N01.DI.SIG_FAULT" : Bool AT %DB5033.DBX7.2, 500 ms
   "2910RS001A01N01.DI.EnConfig" : Bool AT %DB5033.DBX7.3, 500 ms
   "2910RS001A01N01.DI.AEN" : Bool AT %DB5033.DBX7.4, 500 ms
   "2910RS001A01N01.DI.AL_SUPR" : Bool AT %DB5033.DBX7.5, 500 ms
   "2910RS001A01N01.Q.PV_NORM" : Real AT %DB5033.DBD8, 500 ms
   "2910RS001A01N01.Q.PV_SCAL" : Real AT %DB5033.DBD12, 500 ms
   "2910RS001A01N01.ParentInfo" : TextRef, internal   // Имя родителя для попап окна, вкладка инфо. При експорте из ECS через скрипт заполняется автоматически, если теги копируются в ручную то требуется в ручную задатать свойство Start Value

HMI tags "2915RS001A01F01"
   "2915RS001A01F01.MSW" : 52809b66-421d-457f-8884-6f7a49d4e247 AT %DB5036.DBX18.0, 500 ms
   "2915RS001A01F01.DefaultText" : TextRef, internal   // Заголовок POPUP окна. При експорте из ECS через скрипт заполняется автоматически, если теги копируются в ручную то требуется в ручную задатать свойство Start Value
   "2915RS001A01F01.BlockInfo" : Array [0..2] of Int AT %DB5036.DBX38.0, 500 ms
   "2915RS001A01F01.StatusWork" : Int AT %DB5036.DBW242, 500 ms
   "2915RS001A01F01.FP_PARAM.DampingTime" : Int AT %DB5036.DBW50, 500 ms
   "2915RS001A01F01.FP_PARAM.Force_Value" : Real AT %DB5036.DBD52, 500 ms
   "2915RS001A01F01.FP_PARAM.Scale_Min" : Real AT %DB5036.DBD56, 500 ms
   "2915RS001A01F01.FP_PARAM.Scale_Max" : Real AT %DB5036.DBD60, 500 ms
   "2915RS001A01F01.FP_PARAM.Gradient" : Real AT %DB5036.DBD64, 500 ms
   "2915RS001A01F01.FP_PARAM.Grad_Pos" : Real AT %DB5036.DBD68, 500 ms
   "2915RS001A01F01.FP_PARAM.Grad_Neg" : Real AT %DB5036.DBD72, 500 ms
   "2915RS001A01F01.FP_PARAM.Grad_X" : Real AT %DB5036.DBD76, 500 ms
   "2915RS001A01F01.FP_PARAM.Gradient_Time_Pre" : Int AT %DB5036.DBW80, 500 ms
   "2915RS001A01F01.FP_PARAM.Gradient_Time_ACC" : Int AT %DB5036.DBW82, 500 ms
   "2915RS001A01F01.FP_PARAM.Alarm_Hyst" : Real AT %DB5036.DBD84, 500 ms
   "2915RS001A01F01.FP_PARAM.AlarmLimit_H3" : Real AT %DB5036.DBD88, 500 ms
   "2915RS001A01F01.FP_PARAM.AlarmLimit_H2" : Real AT %DB5036.DBD92, 500 ms
   "2915RS001A01F01.FP_PARAM.AlarmLimit_H1" : Real AT %DB5036.DBD96, 500 ms
   "2915RS001A01F01.FP_PARAM.AlarmLimit_L1" : Real AT %DB5036.DBD100, 500 ms
   "2915RS001A01F01.FP_PARAM.AlarmLimit_L2" : Real AT %DB5036.DBD104, 500 ms
   "2915RS001A01F01.FP_PARAM.AlarmLimit_L3" : Real AT %DB5036.DBD108, 500 ms
   "2915RS001A01F01.FP_PARAM.AlarmDelay_H3_Pre" : Int AT %DB5036.DBW112, 500 ms
   "2915RS001A01F01.FP_PARAM.AlarmDelay_H3_Acc" : Int AT %DB5036.DBW114, 500 ms
   "2915RS001A01F01.FP_PARAM.AlarmDelay_H2_Pre" : Int AT %DB5036.DBW116, 500 ms
   "2915RS001A01F01.FP_PARAM.AlarmDelay_H2_Acc" : Int AT %DB5036.DBW118, 500 ms
   "2915RS001A01F01.FP_PARAM.AlarmDelay_H1_Pre" : Int AT %DB5036.DBW120, 500 ms
   "2915RS001A01F01.FP_PARAM.AlarmDelay_H1_Acc" : Int AT %DB5036.DBW122, 500 ms
   "2915RS001A01F01.FP_PARAM.AlarmDelay_L1_Pre" : Int AT %DB5036.DBW124, 500 ms
   "2915RS001A01F01.FP_PARAM.AlarmDelay_L1_Acc" : Int AT %DB5036.DBW126, 500 ms
   "2915RS001A01F01.FP_PARAM.AlarmDelay_L2_Pre" : Int AT %DB5036.DBW128, 500 ms
   "2915RS001A01F01.FP_PARAM.AlarmDelay_L2_Acc" : Int AT %DB5036.DBW130, 500 ms
   "2915RS001A01F01.FP_PARAM.AlarmDelay_L3_Pre" : Int AT %DB5036.DBW132, 500 ms
   "2915RS001A01F01.FP_PARAM.AlarmDelay_L3_Acc" : Int AT %DB5036.DBW134, 500 ms
   "2915RS001A01F01.FP_PARAM.OpenLoopDelay_Pre" : Int AT %DB5036.DBW136, 500 ms
   "2915RS001A01F01.FP_PARAM.OpenLoopDelay_Acc" : Int AT %DB5036.DBW138, 500 ms
   "2915RS001A01F01.FP_PARAM.OverRangeDelay_Pre" : Int AT %DB5036.DBW140, 500 ms
   "2915RS001A01F01.FP_PARAM.OverRangeDelay_Acc" : Int AT %DB5036.DBW142, 500 ms
   "2915RS001A01F01.FP_PARAM.AuxLimit_H2_Value" : Real AT %DB5036.DBD144, 500 ms
   "2915RS001A01F01.FP_PARAM.AuxLimit_H1_Value" : Real AT %DB5036.DBD148, 500 ms
   "2915RS001A01F01.FP_PARAM.AuxLimit_L2_Value" : Real AT %DB5036.DBD152, 500 ms
   "2915RS001A01F01.FP_PARAM.AuxLimit_L1_Value" : Real AT %DB5036.DBD156, 500 ms
   "2915RS001A01F01.Unit" : TextRef, internal   // Еденицы измерения При експорте из ECS через скрипт заполняется автоматически, если теги копируются в ручную то требуется задатать свойство Text
   "2915RS001A01F01.Decimals" : TextRef, internal   // Формат отображения При експорте из ECS через скрипт, заполняется автоматически. Если теги копируются в ручную то требуется задатать свойство Text s999999.9
   "2915RS001A01F01.FP_EN.Square" : Bool AT %DB5036.DBX46.0, 500 ms
   "2915RS001A01F01.FP_EN.SquareRoot" : Bool AT %DB5036.DBX46.1, 500 ms
   "2915RS001A01F01.FP_EN.ParentSupress" : Bool AT %DB5036.DBX46.2, 500 ms
   "2915RS001A01F01.FP_EN.ParentSupressUnit" : Bool AT %DB5036.DBX46.3, 500 ms
   "2915RS001A01F01.FP_EN.Force" : Bool AT %DB5036.DBX46.4, 500 ms
   "2915RS001A01F01.FP_EN.Damping" : Bool AT %DB5036.DBX46.5, 500 ms
   "2915RS001A01F01.FP_EN.Gradient_Pos" : Bool AT %DB5036.DBX46.6, 500 ms
   "2915RS001A01F01.FP_EN.Gradient_Neg" : Bool AT %DB5036.DBX46.7, 500 ms
   "2915RS001A01F01.FP_EN.Hysteresis" : Bool AT %DB5036.DBX47.0, 500 ms
   "2915RS001A01F01.FP_EN.Alarm_H3" : Bool AT %DB5036.DBX47.1, 500 ms
   "2915RS001A01F01.FP_EN.Alarm_H2" : Bool AT %DB5036.DBX47.2, 500 ms
   "2915RS001A01F01.FP_EN.Alarm_H1" : Bool AT %DB5036.DBX47.3, 500 ms
   "2915RS001A01F01.FP_EN.Alarm_L1" : Bool AT %DB5036.DBX47.4, 500 ms
   "2915RS001A01F01.FP_EN.Alarm_L2" : Bool AT %DB5036.DBX47.5, 500 ms
   "2915RS001A01F01.FP_EN.Alarm_L3" : Bool AT %DB5036.DBX47.6, 500 ms
   "2915RS001A01F01.FP_EN.AlarmDelay_H3" : Bool AT %DB5036.DBX47.7, 500 ms
   "2915RS001A01F01.FP_EN.AlarmDelay_H2" : Bool AT %DB5036.DBX48.0, 500 ms
   "2915RS001A01F01.FP_EN.AlarmDelay_H1" : Bool AT %DB5036.DBX48.1, 500 ms
   "2915RS001A01F01.FP_EN.AlarmDelay_L1" : Bool AT %DB5036.DBX48.2, 500 ms
   "2915RS001A01F01.FP_EN.AlarmDelay_L2" : Bool AT %DB5036.DBX48.3, 500 ms
   "2915RS001A01F01.FP_EN.AlarmDelay_L3" : Bool AT %DB5036.DBX48.4, 500 ms
   "2915RS001A01F01.FP_EN.ROC_Warn" : Bool AT %DB5036.DBX48.5, 500 ms
   "2915RS001A01F01.FP_EN.U_Range_Warn" : Bool AT %DB5036.DBX48.6, 500 ms
   "2915RS001A01F01.FP_EN.O_Range_Warn" : Bool AT %DB5036.DBX48.7, 500 ms
   "2915RS001A01F01.trend_tag_name" : TextRef, internal   // Еденицы измерения При експорте из ECS через скрипт - заполняется автоматически, если теги копируются в ручную то требуется задатать свойство Text - имя тега для тренда
   "2915RS001A01F01.DQ.AL_H3" : Bool AT %DB5036.DBX16.0, 500 ms
   "2915RS001A01F01.DQ.AL_H2" : Bool AT %DB5036.DBX16.1, 500 ms
   "2915RS001A01F01.DQ.AL_H1" : Bool AT %DB5036.DBX16.2, 500 ms
   "2915RS001A01F01.DQ.AL_L1" : Bool AT %DB5036.DBX16.3, 500 ms
   "2915RS001A01F01.DQ.AL_L2" : Bool AT %DB5036.DBX16.4, 500 ms
   "2915RS001A01F01.DQ.AL_L3" : Bool AT %DB5036.DBX16.5, 500 ms
   "2915RS001A01F01.DQ.SIG_OK" : Bool AT %DB5036.DBX16.6, 500 ms
   "2915RS001A01F01.DQ.LIM_H2" : Bool AT %DB5036.DBX16.7, 500 ms
   "2915RS001A01F01.DQ.LIM_H1" : Bool AT %DB5036.DBX17.0, 500 ms
   "2915RS001A01F01.DQ.LIM_L1" : Bool AT %DB5036.DBX17.1, 500 ms
   "2915RS001A01F01.DQ.LIM_L2" : Bool AT %DB5036.DBX17.2, 500 ms
   "2915RS001A01F01.DQ.GR_P" : Bool AT %DB5036.DBX17.3, 500 ms
   "2915RS001A01F01.DQ.GR_N" : Bool AT %DB5036.DBX17.4, 500 ms
   "2915RS001A01F01.I.IN" : Real AT %DB5036.DBD2, 500 ms
   "2915RS001A01F01.I.SIG_TYPE" : Int AT %DB5036.DBW0, 500 ms
   "2915RS001A01F01.I.FI_BUS" : Byte AT %DB5036.DBB6, 500 ms
   "2915RS001A01F01.DI.U_RANGE" : Bool AT %DB5036.DBX7.0, 500 ms
   "2915RS001A01F01.DI.O_RANGE" : Bool AT %DB5036.DBX7.1, 500 ms
   "2915RS001A01F01.DI.SIG_FAULT" : Bool AT %DB5036.DBX7.2, 500 ms
   "2915RS001A01F01.DI.EnConfig" : Bool AT %DB5036.DBX7.3, 500 ms
   "2915RS001A01F01.DI.AEN" : Bool AT %DB5036.DBX7.4, 500 ms
   "2915RS001A01F01.DI.AL_SUPR" : Bool AT %DB5036.DBX7.5, 500 ms
   "2915RS001A01F01.Q.PV_NORM" : Real AT %DB5036.DBD8, 500 ms
   "2915RS001A01F01.Q.PV_SCAL" : Real AT %DB5036.DBD12, 500 ms
   "2915RS001A01F01.ParentInfo" : TextRef, internal   // Имя родителя для попап окна, вкладка инфо. При експорте из ECS через скрипт заполняется автоматически, если теги копируются в ручную то требуется в ручную задатать свойство Start Value

HMI tags "2915RS001A01F02"
   "2915RS001A01F02.MSW" : 52809b66-421d-457f-8884-6f7a49d4e247 AT %DB5037.DBX18.0, 500 ms
   "2915RS001A01F02.DefaultText" : TextRef, internal   // Заголовок POPUP окна. При експорте из ECS через скрипт заполняется автоматически, если теги копируются в ручную то требуется в ручную задатать свойство Start Value
   "2915RS001A01F02.BlockInfo" : Array [0..2] of Int AT %DB5037.DBX38.0, 500 ms
   "2915RS001A01F02.StatusWork" : Int AT %DB5037.DBW242, 500 ms
   "2915RS001A01F02.FP_PARAM.DampingTime" : Int AT %DB5037.DBW50, 500 ms
   "2915RS001A01F02.FP_PARAM.Force_Value" : Real AT %DB5037.DBD52, 500 ms
   "2915RS001A01F02.FP_PARAM.Scale_Min" : Real AT %DB5037.DBD56, 500 ms
   "2915RS001A01F02.FP_PARAM.Scale_Max" : Real AT %DB5037.DBD60, 500 ms
   "2915RS001A01F02.FP_PARAM.Gradient" : Real AT %DB5037.DBD64, 500 ms
   "2915RS001A01F02.FP_PARAM.Grad_Pos" : Real AT %DB5037.DBD68, 500 ms
   "2915RS001A01F02.FP_PARAM.Grad_Neg" : Real AT %DB5037.DBD72, 500 ms
   "2915RS001A01F02.FP_PARAM.Grad_X" : Real AT %DB5037.DBD76, 500 ms
   "2915RS001A01F02.FP_PARAM.Gradient_Time_Pre" : Int AT %DB5037.DBW80, 500 ms
   "2915RS001A01F02.FP_PARAM.Gradient_Time_ACC" : Int AT %DB5037.DBW82, 500 ms
   "2915RS001A01F02.FP_PARAM.Alarm_Hyst" : Real AT %DB5037.DBD84, 500 ms
   "2915RS001A01F02.FP_PARAM.AlarmLimit_H3" : Real AT %DB5037.DBD88, 500 ms
   "2915RS001A01F02.FP_PARAM.AlarmLimit_H2" : Real AT %DB5037.DBD92, 500 ms
   "2915RS001A01F02.FP_PARAM.AlarmLimit_H1" : Real AT %DB5037.DBD96, 500 ms
   "2915RS001A01F02.FP_PARAM.AlarmLimit_L1" : Real AT %DB5037.DBD100, 500 ms
   "2915RS001A01F02.FP_PARAM.AlarmLimit_L2" : Real AT %DB5037.DBD104, 500 ms
   "2915RS001A01F02.FP_PARAM.AlarmLimit_L3" : Real AT %DB5037.DBD108, 500 ms
   "2915RS001A01F02.FP_PARAM.AlarmDelay_H3_Pre" : Int AT %DB5037.DBW112, 500 ms
   "2915RS001A01F02.FP_PARAM.AlarmDelay_H3_Acc" : Int AT %DB5037.DBW114, 500 ms
   "2915RS001A01F02.FP_PARAM.AlarmDelay_H2_Pre" : Int AT %DB5037.DBW116, 500 ms
   "2915RS001A01F02.FP_PARAM.AlarmDelay_H2_Acc" : Int AT %DB5037.DBW118, 500 ms
   "2915RS001A01F02.FP_PARAM.AlarmDelay_H1_Pre" : Int AT %DB5037.DBW120, 500 ms
   "2915RS001A01F02.FP_PARAM.AlarmDelay_H1_Acc" : Int AT %DB5037.DBW122, 500 ms
   "2915RS001A01F02.FP_PARAM.AlarmDelay_L1_Pre" : Int AT %DB5037.DBW124, 500 ms
   "2915RS001A01F02.FP_PARAM.AlarmDelay_L1_Acc" : Int AT %DB5037.DBW126, 500 ms
   "2915RS001A01F02.FP_PARAM.AlarmDelay_L2_Pre" : Int AT %DB5037.DBW128, 500 ms
   "2915RS001A01F02.FP_PARAM.AlarmDelay_L2_Acc" : Int AT %DB5037.DBW130, 500 ms
   "2915RS001A01F02.FP_PARAM.AlarmDelay_L3_Pre" : Int AT %DB5037.DBW132, 500 ms
   "2915RS001A01F02.FP_PARAM.AlarmDelay_L3_Acc" : Int AT %DB5037.DBW134, 500 ms
   "2915RS001A01F02.FP_PARAM.OpenLoopDelay_Pre" : Int AT %DB5037.DBW136, 500 ms
   "2915RS001A01F02.FP_PARAM.OpenLoopDelay_Acc" : Int AT %DB5037.DBW138, 500 ms
   "2915RS001A01F02.FP_PARAM.OverRangeDelay_Pre" : Int AT %DB5037.DBW140, 500 ms
   "2915RS001A01F02.FP_PARAM.OverRangeDelay_Acc" : Int AT %DB5037.DBW142, 500 ms
   "2915RS001A01F02.FP_PARAM.AuxLimit_H2_Value" : Real AT %DB5037.DBD144, 500 ms
   "2915RS001A01F02.FP_PARAM.AuxLimit_H1_Value" : Real AT %DB5037.DBD148, 500 ms
   "2915RS001A01F02.FP_PARAM.AuxLimit_L2_Value" : Real AT %DB5037.DBD152, 500 ms
   "2915RS001A01F02.FP_PARAM.AuxLimit_L1_Value" : Real AT %DB5037.DBD156, 500 ms
   "2915RS001A01F02.Unit" : TextRef, internal   // Еденицы измерения При експорте из ECS через скрипт заполняется автоматически, если теги копируются в ручную то требуется задатать свойство Text
   "2915RS001A01F02.Decimals" : TextRef, internal   // Формат отображения При експорте из ECS через скрипт, заполняется автоматически. Если теги копируются в ручную то требуется задатать свойство Text s999999.9
   "2915RS001A01F02.FP_EN.Square" : Bool AT %DB5037.DBX46.0, 500 ms
   "2915RS001A01F02.FP_EN.SquareRoot" : Bool AT %DB5037.DBX46.1, 500 ms
   "2915RS001A01F02.FP_EN.ParentSupress" : Bool AT %DB5037.DBX46.2, 500 ms
   "2915RS001A01F02.FP_EN.ParentSupressUnit" : Bool AT %DB5037.DBX46.3, 500 ms
   "2915RS001A01F02.FP_EN.Force" : Bool AT %DB5037.DBX46.4, 500 ms
   "2915RS001A01F02.FP_EN.Damping" : Bool AT %DB5037.DBX46.5, 500 ms
   "2915RS001A01F02.FP_EN.Gradient_Pos" : Bool AT %DB5037.DBX46.6, 500 ms
   "2915RS001A01F02.FP_EN.Gradient_Neg" : Bool AT %DB5037.DBX46.7, 500 ms
   "2915RS001A01F02.FP_EN.Hysteresis" : Bool AT %DB5037.DBX47.0, 500 ms
   "2915RS001A01F02.FP_EN.Alarm_H3" : Bool AT %DB5037.DBX47.1, 500 ms
   "2915RS001A01F02.FP_EN.Alarm_H2" : Bool AT %DB5037.DBX47.2, 500 ms
   "2915RS001A01F02.FP_EN.Alarm_H1" : Bool AT %DB5037.DBX47.3, 500 ms
   "2915RS001A01F02.FP_EN.Alarm_L1" : Bool AT %DB5037.DBX47.4, 500 ms
   "2915RS001A01F02.FP_EN.Alarm_L2" : Bool AT %DB5037.DBX47.5, 500 ms
   "2915RS001A01F02.FP_EN.Alarm_L3" : Bool AT %DB5037.DBX47.6, 500 ms
   "2915RS001A01F02.FP_EN.AlarmDelay_H3" : Bool AT %DB5037.DBX47.7, 500 ms
   "2915RS001A01F02.FP_EN.AlarmDelay_H2" : Bool AT %DB5037.DBX48.0, 500 ms
   "2915RS001A01F02.FP_EN.AlarmDelay_H1" : Bool AT %DB5037.DBX48.1, 500 ms
   "2915RS001A01F02.FP_EN.AlarmDelay_L1" : Bool AT %DB5037.DBX48.2, 500 ms
   "2915RS001A01F02.FP_EN.AlarmDelay_L2" : Bool AT %DB5037.DBX48.3, 500 ms
   "2915RS001A01F02.FP_EN.AlarmDelay_L3" : Bool AT %DB5037.DBX48.4, 500 ms
   "2915RS001A01F02.FP_EN.ROC_Warn" : Bool AT %DB5037.DBX48.5, 500 ms
   "2915RS001A01F02.FP_EN.U_Range_Warn" : Bool AT %DB5037.DBX48.6, 500 ms
   "2915RS001A01F02.FP_EN.O_Range_Warn" : Bool AT %DB5037.DBX48.7, 500 ms
   "2915RS001A01F02.trend_tag_name" : TextRef, internal   // Еденицы измерения При експорте из ECS через скрипт - заполняется автоматически, если теги копируются в ручную то требуется задатать свойство Text - имя тега для тренда
   "2915RS001A01F02.DQ.AL_H3" : Bool AT %DB5037.DBX16.0, 500 ms
   "2915RS001A01F02.DQ.AL_H2" : Bool AT %DB5037.DBX16.1, 500 ms
   "2915RS001A01F02.DQ.AL_H1" : Bool AT %DB5037.DBX16.2, 500 ms
   "2915RS001A01F02.DQ.AL_L1" : Bool AT %DB5037.DBX16.3, 500 ms
   "2915RS001A01F02.DQ.AL_L2" : Bool AT %DB5037.DBX16.4, 500 ms
   "2915RS001A01F02.DQ.AL_L3" : Bool AT %DB5037.DBX16.5, 500 ms
   "2915RS001A01F02.DQ.SIG_OK" : Bool AT %DB5037.DBX16.6, 500 ms
   "2915RS001A01F02.DQ.LIM_H2" : Bool AT %DB5037.DBX16.7, 500 ms
   "2915RS001A01F02.DQ.LIM_H1" : Bool AT %DB5037.DBX17.0, 500 ms
   "2915RS001A01F02.DQ.LIM_L1" : Bool AT %DB5037.DBX17.1, 500 ms
   "2915RS001A01F02.DQ.LIM_L2" : Bool AT %DB5037.DBX17.2, 500 ms
   "2915RS001A01F02.DQ.GR_P" : Bool AT %DB5037.DBX17.3, 500 ms
   "2915RS001A01F02.DQ.GR_N" : Bool AT %DB5037.DBX17.4, 500 ms
   "2915RS001A01F02.I.IN" : Real AT %DB5037.DBD2, 500 ms
   "2915RS001A01F02.I.SIG_TYPE" : Int AT %DB5037.DBW0, 500 ms
   "2915RS001A01F02.I.FI_BUS" : Byte AT %DB5037.DBB6, 500 ms
   "2915RS001A01F02.DI.U_RANGE" : Bool AT %DB5037.DBX7.0, 500 ms
   "2915RS001A01F02.DI.O_RANGE" : Bool AT %DB5037.DBX7.1, 500 ms
   "2915RS001A01F02.DI.SIG_FAULT" : Bool AT %DB5037.DBX7.2, 500 ms
   "2915RS001A01F02.DI.EnConfig" : Bool AT %DB5037.DBX7.3, 500 ms
   "2915RS001A01F02.DI.AEN" : Bool AT %DB5037.DBX7.4, 500 ms
   "2915RS001A01F02.DI.AL_SUPR" : Bool AT %DB5037.DBX7.5, 500 ms
   "2915RS001A01F02.Q.PV_NORM" : Real AT %DB5037.DBD8, 500 ms
   "2915RS001A01F02.Q.PV_SCAL" : Real AT %DB5037.DBD12, 500 ms
   "2915RS001A01F02.ParentInfo" : TextRef, internal   // Имя родителя для попап окна, вкладка инфо. При експорте из ECS через скрипт заполняется автоматически, если теги копируются в ручную то требуется в ручную задатать свойство Start Value

HMI tags "2915RS001A01F03"
   "2915RS001A01F03.MSW" : 52809b66-421d-457f-8884-6f7a49d4e247 AT %DB5038.DBX18.0, 500 ms
   "2915RS001A01F03.DefaultText" : TextRef, internal   // Заголовок POPUP окна. При експорте из ECS через скрипт заполняется автоматически, если теги копируются в ручную то требуется в ручную задатать свойство Start Value
   "2915RS001A01F03.BlockInfo" : Array [0..2] of Int AT %DB5038.DBX38.0, 500 ms
   "2915RS001A01F03.StatusWork" : Int AT %DB5038.DBW242, 500 ms
   "2915RS001A01F03.FP_PARAM.DampingTime" : Int AT %DB5038.DBW50, 500 ms
   "2915RS001A01F03.FP_PARAM.Force_Value" : Real AT %DB5038.DBD52, 500 ms
   "2915RS001A01F03.FP_PARAM.Scale_Min" : Real AT %DB5038.DBD56, 500 ms
   "2915RS001A01F03.FP_PARAM.Scale_Max" : Real AT %DB5038.DBD60, 500 ms
   "2915RS001A01F03.FP_PARAM.Gradient" : Real AT %DB5038.DBD64, 500 ms
   "2915RS001A01F03.FP_PARAM.Grad_Pos" : Real AT %DB5038.DBD68, 500 ms
   "2915RS001A01F03.FP_PARAM.Grad_Neg" : Real AT %DB5038.DBD72, 500 ms
   "2915RS001A01F03.FP_PARAM.Grad_X" : Real AT %DB5038.DBD76, 500 ms
   "2915RS001A01F03.FP_PARAM.Gradient_Time_Pre" : Int AT %DB5038.DBW80, 500 ms
   "2915RS001A01F03.FP_PARAM.Gradient_Time_ACC" : Int AT %DB5038.DBW82, 500 ms
   "2915RS001A01F03.FP_PARAM.Alarm_Hyst" : Real AT %DB5038.DBD84, 500 ms
   "2915RS001A01F03.FP_PARAM.AlarmLimit_H3" : Real AT %DB5038.DBD88, 500 ms
   "2915RS001A01F03.FP_PARAM.AlarmLimit_H2" : Real AT %DB5038.DBD92, 500 ms
   "2915RS001A01F03.FP_PARAM.AlarmLimit_H1" : Real AT %DB5038.DBD96, 500 ms
   "2915RS001A01F03.FP_PARAM.AlarmLimit_L1" : Real AT %DB5038.DBD100, 500 ms
   "2915RS001A01F03.FP_PARAM.AlarmLimit_L2" : Real AT %DB5038.DBD104, 500 ms
   "2915RS001A01F03.FP_PARAM.AlarmLimit_L3" : Real AT %DB5038.DBD108, 500 ms
   "2915RS001A01F03.FP_PARAM.AlarmDelay_H3_Pre" : Int AT %DB5038.DBW112, 500 ms
   "2915RS001A01F03.FP_PARAM.AlarmDelay_H3_Acc" : Int AT %DB5038.DBW114, 500 ms
   "2915RS001A01F03.FP_PARAM.AlarmDelay_H2_Pre" : Int AT %DB5038.DBW116, 500 ms
   "2915RS001A01F03.FP_PARAM.AlarmDelay_H2_Acc" : Int AT %DB5038.DBW118, 500 ms
   "2915RS001A01F03.FP_PARAM.AlarmDelay_H1_Pre" : Int AT %DB5038.DBW120, 500 ms
   "2915RS001A01F03.FP_PARAM.AlarmDelay_H1_Acc" : Int AT %DB5038.DBW122, 500 ms
   "2915RS001A01F03.FP_PARAM.AlarmDelay_L1_Pre" : Int AT %DB5038.DBW124, 500 ms
   "2915RS001A01F03.FP_PARAM.AlarmDelay_L1_Acc" : Int AT %DB5038.DBW126, 500 ms
   "2915RS001A01F03.FP_PARAM.AlarmDelay_L2_Pre" : Int AT %DB5038.DBW128, 500 ms
   "2915RS001A01F03.FP_PARAM.AlarmDelay_L2_Acc" : Int AT %DB5038.DBW130, 500 ms
   "2915RS001A01F03.FP_PARAM.AlarmDelay_L3_Pre" : Int AT %DB5038.DBW132, 500 ms
   "2915RS001A01F03.FP_PARAM.AlarmDelay_L3_Acc" : Int AT %DB5038.DBW134, 500 ms
   "2915RS001A01F03.FP_PARAM.OpenLoopDelay_Pre" : Int AT %DB5038.DBW136, 500 ms
   "2915RS001A01F03.FP_PARAM.OpenLoopDelay_Acc" : Int AT %DB5038.DBW138, 500 ms
   "2915RS001A01F03.FP_PARAM.OverRangeDelay_Pre" : Int AT %DB5038.DBW140, 500 ms
   "2915RS001A01F03.FP_PARAM.OverRangeDelay_Acc" : Int AT %DB5038.DBW142, 500 ms
   "2915RS001A01F03.FP_PARAM.AuxLimit_H2_Value" : Real AT %DB5038.DBD144, 500 ms
   "2915RS001A01F03.FP_PARAM.AuxLimit_H1_Value" : Real AT %DB5038.DBD148, 500 ms
   "2915RS001A01F03.FP_PARAM.AuxLimit_L2_Value" : Real AT %DB5038.DBD152, 500 ms
   "2915RS001A01F03.FP_PARAM.AuxLimit_L1_Value" : Real AT %DB5038.DBD156, 500 ms
   "2915RS001A01F03.Unit" : TextRef, internal   // Еденицы измерения При експорте из ECS через скрипт заполняется автоматически, если теги копируются в ручную то требуется задатать свойство Text
   "2915RS001A01F03.Decimals" : TextRef, internal   // Формат отображения При експорте из ECS через скрипт, заполняется автоматически. Если теги копируются в ручную то требуется задатать свойство Text s999999.9
   "2915RS001A01F03.FP_EN.Square" : Bool AT %DB5038.DBX46.0, 500 ms
   "2915RS001A01F03.FP_EN.SquareRoot" : Bool AT %DB5038.DBX46.1, 500 ms
   "2915RS001A01F03.FP_EN.ParentSupress" : Bool AT %DB5038.DBX46.2, 500 ms
   "2915RS001A01F03.FP_EN.ParentSupressUnit" : Bool AT %DB5038.DBX46.3, 500 ms
   "2915RS001A01F03.FP_EN.Force" : Bool AT %DB5038.DBX46.4, 500 ms
   "2915RS001A01F03.FP_EN.Damping" : Bool AT %DB5038.DBX46.5, 500 ms
   "2915RS001A01F03.FP_EN.Gradient_Pos" : Bool AT %DB5038.DBX46.6, 500 ms
   "2915RS001A01F03.FP_EN.Gradient_Neg" : Bool AT %DB5038.DBX46.7, 500 ms
   "2915RS001A01F03.FP_EN.Hysteresis" : Bool AT %DB5038.DBX47.0, 500 ms
   "2915RS001A01F03.FP_EN.Alarm_H3" : Bool AT %DB5038.DBX47.1, 500 ms
   "2915RS001A01F03.FP_EN.Alarm_H2" : Bool AT %DB5038.DBX47.2, 500 ms
   "2915RS001A01F03.FP_EN.Alarm_H1" : Bool AT %DB5038.DBX47.3, 500 ms
   "2915RS001A01F03.FP_EN.Alarm_L1" : Bool AT %DB5038.DBX47.4, 500 ms
   "2915RS001A01F03.FP_EN.Alarm_L2" : Bool AT %DB5038.DBX47.5, 500 ms
   "2915RS001A01F03.FP_EN.Alarm_L3" : Bool AT %DB5038.DBX47.6, 500 ms
   "2915RS001A01F03.FP_EN.AlarmDelay_H3" : Bool AT %DB5038.DBX47.7, 500 ms
   "2915RS001A01F03.FP_EN.AlarmDelay_H2" : Bool AT %DB5038.DBX48.0, 500 ms
   "2915RS001A01F03.FP_EN.AlarmDelay_H1" : Bool AT %DB5038.DBX48.1, 500 ms
   "2915RS001A01F03.FP_EN.AlarmDelay_L1" : Bool AT %DB5038.DBX48.2, 500 ms
   "2915RS001A01F03.FP_EN.AlarmDelay_L2" : Bool AT %DB5038.DBX48.3, 500 ms
   "2915RS001A01F03.FP_EN.AlarmDelay_L3" : Bool AT %DB5038.DBX48.4, 500 ms
   "2915RS001A01F03.FP_EN.ROC_Warn" : Bool AT %DB5038.DBX48.5, 500 ms
   "2915RS001A01F03.FP_EN.U_Range_Warn" : Bool AT %DB5038.DBX48.6, 500 ms
   "2915RS001A01F03.FP_EN.O_Range_Warn" : Bool AT %DB5038.DBX48.7, 500 ms
   "2915RS001A01F03.trend_tag_name" : TextRef, internal   // Еденицы измерения При експорте из ECS через скрипт - заполняется автоматически, если теги копируются в ручную то требуется задатать свойство Text - имя тега для тренда
   "2915RS001A01F03.DQ.AL_H3" : Bool AT %DB5038.DBX16.0, 500 ms
   "2915RS001A01F03.DQ.AL_H2" : Bool AT %DB5038.DBX16.1, 500 ms
   "2915RS001A01F03.DQ.AL_H1" : Bool AT %DB5038.DBX16.2, 500 ms
   "2915RS001A01F03.DQ.AL_L1" : Bool AT %DB5038.DBX16.3, 500 ms
   "2915RS001A01F03.DQ.AL_L2" : Bool AT %DB5038.DBX16.4, 500 ms
   "2915RS001A01F03.DQ.AL_L3" : Bool AT %DB5038.DBX16.5, 500 ms
   "2915RS001A01F03.DQ.SIG_OK" : Bool AT %DB5038.DBX16.6, 500 ms
   "2915RS001A01F03.DQ.LIM_H2" : Bool AT %DB5038.DBX16.7, 500 ms
   "2915RS001A01F03.DQ.LIM_H1" : Bool AT %DB5038.DBX17.0, 500 ms
   "2915RS001A01F03.DQ.LIM_L1" : Bool AT %DB5038.DBX17.1, 500 ms
   "2915RS001A01F03.DQ.LIM_L2" : Bool AT %DB5038.DBX17.2, 500 ms
   "2915RS001A01F03.DQ.GR_P" : Bool AT %DB5038.DBX17.3, 500 ms
   "2915RS001A01F03.DQ.GR_N" : Bool AT %DB5038.DBX17.4, 500 ms
   "2915RS001A01F03.I.IN" : Real AT %DB5038.DBD2, 500 ms
   "2915RS001A01F03.I.SIG_TYPE" : Int AT %DB5038.DBW0, 500 ms
   "2915RS001A01F03.I.FI_BUS" : Byte AT %DB5038.DBB6, 500 ms
   "2915RS001A01F03.DI.U_RANGE" : Bool AT %DB5038.DBX7.0, 500 ms
   "2915RS001A01F03.DI.O_RANGE" : Bool AT %DB5038.DBX7.1, 500 ms
   "2915RS001A01F03.DI.SIG_FAULT" : Bool AT %DB5038.DBX7.2, 500 ms
   "2915RS001A01F03.DI.EnConfig" : Bool AT %DB5038.DBX7.3, 500 ms
   "2915RS001A01F03.DI.AEN" : Bool AT %DB5038.DBX7.4, 500 ms
   "2915RS001A01F03.DI.AL_SUPR" : Bool AT %DB5038.DBX7.5, 500 ms
   "2915RS001A01F03.Q.PV_NORM" : Real AT %DB5038.DBD8, 500 ms
   "2915RS001A01F03.Q.PV_SCAL" : Real AT %DB5038.DBD12, 500 ms
   "2915RS001A01F03.ParentInfo" : TextRef, internal   // Имя родителя для попап окна, вкладка инфо. При експорте из ECS через скрипт заполняется автоматически, если теги копируются в ручную то требуется в ручную задатать свойство Start Value

HMI tags "2915RS001A01L01"
   "2915RS001A01L01.MSW" : 52809b66-421d-457f-8884-6f7a49d4e247 AT %DB5039.DBX18.0, 500 ms
   "2915RS001A01L01.DefaultText" : TextRef, internal   // Заголовок POPUP окна. При експорте из ECS через скрипт заполняется автоматически, если теги копируются в ручную то требуется в ручную задатать свойство Start Value
   "2915RS001A01L01.BlockInfo" : Array [0..2] of Int AT %DB5039.DBX38.0, 500 ms
   "2915RS001A01L01.StatusWork" : Int AT %DB5039.DBW242, 500 ms
   "2915RS001A01L01.FP_PARAM.DampingTime" : Int AT %DB5039.DBW50, 500 ms
   "2915RS001A01L01.FP_PARAM.Force_Value" : Real AT %DB5039.DBD52, 500 ms
   "2915RS001A01L01.FP_PARAM.Scale_Min" : Real AT %DB5039.DBD56, 500 ms
   "2915RS001A01L01.FP_PARAM.Scale_Max" : Real AT %DB5039.DBD60, 500 ms
   "2915RS001A01L01.FP_PARAM.Gradient" : Real AT %DB5039.DBD64, 500 ms
   "2915RS001A01L01.FP_PARAM.Grad_Pos" : Real AT %DB5039.DBD68, 500 ms
   "2915RS001A01L01.FP_PARAM.Grad_Neg" : Real AT %DB5039.DBD72, 500 ms
   "2915RS001A01L01.FP_PARAM.Grad_X" : Real AT %DB5039.DBD76, 500 ms
   "2915RS001A01L01.FP_PARAM.Gradient_Time_Pre" : Int AT %DB5039.DBW80, 500 ms
   "2915RS001A01L01.FP_PARAM.Gradient_Time_ACC" : Int AT %DB5039.DBW82, 500 ms
   "2915RS001A01L01.FP_PARAM.Alarm_Hyst" : Real AT %DB5039.DBD84, 500 ms
   "2915RS001A01L01.FP_PARAM.AlarmLimit_H3" : Real AT %DB5039.DBD88, 500 ms
   "2915RS001A01L01.FP_PARAM.AlarmLimit_H2" : Real AT %DB5039.DBD92, 500 ms
   "2915RS001A01L01.FP_PARAM.AlarmLimit_H1" : Real AT %DB5039.DBD96, 500 ms
   "2915RS001A01L01.FP_PARAM.AlarmLimit_L1" : Real AT %DB5039.DBD100, 500 ms
   "2915RS001A01L01.FP_PARAM.AlarmLimit_L2" : Real AT %DB5039.DBD104, 500 ms
   "2915RS001A01L01.FP_PARAM.AlarmLimit_L3" : Real AT %DB5039.DBD108, 500 ms
   "2915RS001A01L01.FP_PARAM.AlarmDelay_H3_Pre" : Int AT %DB5039.DBW112, 500 ms
   "2915RS001A01L01.FP_PARAM.AlarmDelay_H3_Acc" : Int AT %DB5039.DBW114, 500 ms
   "2915RS001A01L01.FP_PARAM.AlarmDelay_H2_Pre" : Int AT %DB5039.DBW116, 500 ms
   "2915RS001A01L01.FP_PARAM.AlarmDelay_H2_Acc" : Int AT %DB5039.DBW118, 500 ms
   "2915RS001A01L01.FP_PARAM.AlarmDelay_H1_Pre" : Int AT %DB5039.DBW120, 500 ms
   "2915RS001A01L01.FP_PARAM.AlarmDelay_H1_Acc" : Int AT %DB5039.DBW122, 500 ms
   "2915RS001A01L01.FP_PARAM.AlarmDelay_L1_Pre" : Int AT %DB5039.DBW124, 500 ms
   "2915RS001A01L01.FP_PARAM.AlarmDelay_L1_Acc" : Int AT %DB5039.DBW126, 500 ms
   "2915RS001A01L01.FP_PARAM.AlarmDelay_L2_Pre" : Int AT %DB5039.DBW128, 500 ms
   "2915RS001A01L01.FP_PARAM.AlarmDelay_L2_Acc" : Int AT %DB5039.DBW130, 500 ms
   "2915RS001A01L01.FP_PARAM.AlarmDelay_L3_Pre" : Int AT %DB5039.DBW132, 500 ms
   "2915RS001A01L01.FP_PARAM.AlarmDelay_L3_Acc" : Int AT %DB5039.DBW134, 500 ms
   "2915RS001A01L01.FP_PARAM.OpenLoopDelay_Pre" : Int AT %DB5039.DBW136, 500 ms
   "2915RS001A01L01.FP_PARAM.OpenLoopDelay_Acc" : Int AT %DB5039.DBW138, 500 ms
   "2915RS001A01L01.FP_PARAM.OverRangeDelay_Pre" : Int AT %DB5039.DBW140, 500 ms
   "2915RS001A01L01.FP_PARAM.OverRangeDelay_Acc" : Int AT %DB5039.DBW142, 500 ms
   "2915RS001A01L01.FP_PARAM.AuxLimit_H2_Value" : Real AT %DB5039.DBD144, 500 ms
   "2915RS001A01L01.FP_PARAM.AuxLimit_H1_Value" : Real AT %DB5039.DBD148, 500 ms
   "2915RS001A01L01.FP_PARAM.AuxLimit_L2_Value" : Real AT %DB5039.DBD152, 500 ms
   "2915RS001A01L01.FP_PARAM.AuxLimit_L1_Value" : Real AT %DB5039.DBD156, 500 ms
   "2915RS001A01L01.Unit" : TextRef, internal   // Еденицы измерения При експорте из ECS через скрипт заполняется автоматически, если теги копируются в ручную то требуется задатать свойство Text
   "2915RS001A01L01.Decimals" : TextRef, internal   // Формат отображения При експорте из ECS через скрипт, заполняется автоматически. Если теги копируются в ручную то требуется задатать свойство Text s999999.9
   "2915RS001A01L01.FP_EN.Square" : Bool AT %DB5039.DBX46.0, 500 ms
   "2915RS001A01L01.FP_EN.SquareRoot" : Bool AT %DB5039.DBX46.1, 500 ms
   "2915RS001A01L01.FP_EN.ParentSupress" : Bool AT %DB5039.DBX46.2, 500 ms
   "2915RS001A01L01.FP_EN.ParentSupressUnit" : Bool AT %DB5039.DBX46.3, 500 ms
   "2915RS001A01L01.FP_EN.Force" : Bool AT %DB5039.DBX46.4, 500 ms
   "2915RS001A01L01.FP_EN.Damping" : Bool AT %DB5039.DBX46.5, 500 ms
   "2915RS001A01L01.FP_EN.Gradient_Pos" : Bool AT %DB5039.DBX46.6, 500 ms
   "2915RS001A01L01.FP_EN.Gradient_Neg" : Bool AT %DB5039.DBX46.7, 500 ms
   "2915RS001A01L01.FP_EN.Hysteresis" : Bool AT %DB5039.DBX47.0, 500 ms
   "2915RS001A01L01.FP_EN.Alarm_H3" : Bool AT %DB5039.DBX47.1, 500 ms
   "2915RS001A01L01.FP_EN.Alarm_H2" : Bool AT %DB5039.DBX47.2, 500 ms
   "2915RS001A01L01.FP_EN.Alarm_H1" : Bool AT %DB5039.DBX47.3, 500 ms
   "2915RS001A01L01.FP_EN.Alarm_L1" : Bool AT %DB5039.DBX47.4, 500 ms
   "2915RS001A01L01.FP_EN.Alarm_L2" : Bool AT %DB5039.DBX47.5, 500 ms
   "2915RS001A01L01.FP_EN.Alarm_L3" : Bool AT %DB5039.DBX47.6, 500 ms
   "2915RS001A01L01.FP_EN.AlarmDelay_H3" : Bool AT %DB5039.DBX47.7, 500 ms
   "2915RS001A01L01.FP_EN.AlarmDelay_H2" : Bool AT %DB5039.DBX48.0, 500 ms
   "2915RS001A01L01.FP_EN.AlarmDelay_H1" : Bool AT %DB5039.DBX48.1, 500 ms
   "2915RS001A01L01.FP_EN.AlarmDelay_L1" : Bool AT %DB5039.DBX48.2, 500 ms
   "2915RS001A01L01.FP_EN.AlarmDelay_L2" : Bool AT %DB5039.DBX48.3, 500 ms
   "2915RS001A01L01.FP_EN.AlarmDelay_L3" : Bool AT %DB5039.DBX48.4, 500 ms
   "2915RS001A01L01.FP_EN.ROC_Warn" : Bool AT %DB5039.DBX48.5, 500 ms
   "2915RS001A01L01.FP_EN.U_Range_Warn" : Bool AT %DB5039.DBX48.6, 500 ms
   "2915RS001A01L01.FP_EN.O_Range_Warn" : Bool AT %DB5039.DBX48.7, 500 ms
   "2915RS001A01L01.trend_tag_name" : TextRef, internal   // Еденицы измерения При експорте из ECS через скрипт - заполняется автоматически, если теги копируются в ручную то требуется задатать свойство Text - имя тега для тренда
   "2915RS001A01L01.DQ.AL_H3" : Bool AT %DB5039.DBX16.0, 500 ms
   "2915RS001A01L01.DQ.AL_H2" : Bool AT %DB5039.DBX16.1, 500 ms
   "2915RS001A01L01.DQ.AL_H1" : Bool AT %DB5039.DBX16.2, 500 ms
   "2915RS001A01L01.DQ.AL_L1" : Bool AT %DB5039.DBX16.3, 500 ms
   "2915RS001A01L01.DQ.AL_L2" : Bool AT %DB5039.DBX16.4, 500 ms
   "2915RS001A01L01.DQ.AL_L3" : Bool AT %DB5039.DBX16.5, 500 ms
   "2915RS001A01L01.DQ.SIG_OK" : Bool AT %DB5039.DBX16.6, 500 ms
   "2915RS001A01L01.DQ.LIM_H2" : Bool AT %DB5039.DBX16.7, 500 ms
   "2915RS001A01L01.DQ.LIM_H1" : Bool AT %DB5039.DBX17.0, 500 ms
   "2915RS001A01L01.DQ.LIM_L1" : Bool AT %DB5039.DBX17.1, 500 ms
   "2915RS001A01L01.DQ.LIM_L2" : Bool AT %DB5039.DBX17.2, 500 ms
   "2915RS001A01L01.DQ.GR_P" : Bool AT %DB5039.DBX17.3, 500 ms
   "2915RS001A01L01.DQ.GR_N" : Bool AT %DB5039.DBX17.4, 500 ms
   "2915RS001A01L01.I.IN" : Real AT %DB5039.DBD2, 500 ms
   "2915RS001A01L01.I.SIG_TYPE" : Int AT %DB5039.DBW0, 500 ms
   "2915RS001A01L01.I.FI_BUS" : Byte AT %DB5039.DBB6, 500 ms
   "2915RS001A01L01.DI.U_RANGE" : Bool AT %DB5039.DBX7.0, 500 ms
   "2915RS001A01L01.DI.O_RANGE" : Bool AT %DB5039.DBX7.1, 500 ms
   "2915RS001A01L01.DI.SIG_FAULT" : Bool AT %DB5039.DBX7.2, 500 ms
   "2915RS001A01L01.DI.EnConfig" : Bool AT %DB5039.DBX7.3, 500 ms
   "2915RS001A01L01.DI.AEN" : Bool AT %DB5039.DBX7.4, 500 ms
   "2915RS001A01L01.DI.AL_SUPR" : Bool AT %DB5039.DBX7.5, 500 ms
   "2915RS001A01L01.Q.PV_NORM" : Real AT %DB5039.DBD8, 500 ms
   "2915RS001A01L01.Q.PV_SCAL" : Real AT %DB5039.DBD12, 500 ms
   "2915RS001A01L01.ParentInfo" : TextRef, internal   // Имя родителя для попап окна, вкладка инфо. При експорте из ECS через скрипт заполняется автоматически, если теги копируются в ручную то требуется в ручную задатать свойство Start Value

HMI tags "2915RS001A01L02"
   "2915RS001A01L02.MSW" : 52809b66-421d-457f-8884-6f7a49d4e247 AT %DB5040.DBX18.0, 500 ms
   "2915RS001A01L02.DefaultText" : TextRef, internal   // Заголовок POPUP окна. При експорте из ECS через скрипт заполняется автоматически, если теги копируются в ручную то требуется в ручную задатать свойство Start Value
   "2915RS001A01L02.BlockInfo" : Array [0..2] of Int AT %DB5040.DBX38.0, 500 ms
   "2915RS001A01L02.StatusWork" : Int AT %DB5040.DBW242, 500 ms
   "2915RS001A01L02.FP_PARAM.DampingTime" : Int AT %DB5040.DBW50, 500 ms
   "2915RS001A01L02.FP_PARAM.Force_Value" : Real AT %DB5040.DBD52, 500 ms
   "2915RS001A01L02.FP_PARAM.Scale_Min" : Real AT %DB5040.DBD56, 500 ms
   "2915RS001A01L02.FP_PARAM.Scale_Max" : Real AT %DB5040.DBD60, 500 ms
   "2915RS001A01L02.FP_PARAM.Gradient" : Real AT %DB5040.DBD64, 500 ms
   "2915RS001A01L02.FP_PARAM.Grad_Pos" : Real AT %DB5040.DBD68, 500 ms
   "2915RS001A01L02.FP_PARAM.Grad_Neg" : Real AT %DB5040.DBD72, 500 ms
   "2915RS001A01L02.FP_PARAM.Grad_X" : Real AT %DB5040.DBD76, 500 ms
   "2915RS001A01L02.FP_PARAM.Gradient_Time_Pre" : Int AT %DB5040.DBW80, 500 ms
   "2915RS001A01L02.FP_PARAM.Gradient_Time_ACC" : Int AT %DB5040.DBW82, 500 ms
   "2915RS001A01L02.FP_PARAM.Alarm_Hyst" : Real AT %DB5040.DBD84, 500 ms
   "2915RS001A01L02.FP_PARAM.AlarmLimit_H3" : Real AT %DB5040.DBD88, 500 ms
   "2915RS001A01L02.FP_PARAM.AlarmLimit_H2" : Real AT %DB5040.DBD92, 500 ms
   "2915RS001A01L02.FP_PARAM.AlarmLimit_H1" : Real AT %DB5040.DBD96, 500 ms
   "2915RS001A01L02.FP_PARAM.AlarmLimit_L1" : Real AT %DB5040.DBD100, 500 ms
   "2915RS001A01L02.FP_PARAM.AlarmLimit_L2" : Real AT %DB5040.DBD104, 500 ms
   "2915RS001A01L02.FP_PARAM.AlarmLimit_L3" : Real AT %DB5040.DBD108, 500 ms
   "2915RS001A01L02.FP_PARAM.AlarmDelay_H3_Pre" : Int AT %DB5040.DBW112, 500 ms
   "2915RS001A01L02.FP_PARAM.AlarmDelay_H3_Acc" : Int AT %DB5040.DBW114, 500 ms
   "2915RS001A01L02.FP_PARAM.AlarmDelay_H2_Pre" : Int AT %DB5040.DBW116, 500 ms
   "2915RS001A01L02.FP_PARAM.AlarmDelay_H2_Acc" : Int AT %DB5040.DBW118, 500 ms
   "2915RS001A01L02.FP_PARAM.AlarmDelay_H1_Pre" : Int AT %DB5040.DBW120, 500 ms
   "2915RS001A01L02.FP_PARAM.AlarmDelay_H1_Acc" : Int AT %DB5040.DBW122, 500 ms
   "2915RS001A01L02.FP_PARAM.AlarmDelay_L1_Pre" : Int AT %DB5040.DBW124, 500 ms
   "2915RS001A01L02.FP_PARAM.AlarmDelay_L1_Acc" : Int AT %DB5040.DBW126, 500 ms
   "2915RS001A01L02.FP_PARAM.AlarmDelay_L2_Pre" : Int AT %DB5040.DBW128, 500 ms
   "2915RS001A01L02.FP_PARAM.AlarmDelay_L2_Acc" : Int AT %DB5040.DBW130, 500 ms
   "2915RS001A01L02.FP_PARAM.AlarmDelay_L3_Pre" : Int AT %DB5040.DBW132, 500 ms
   "2915RS001A01L02.FP_PARAM.AlarmDelay_L3_Acc" : Int AT %DB5040.DBW134, 500 ms
   "2915RS001A01L02.FP_PARAM.OpenLoopDelay_Pre" : Int AT %DB5040.DBW136, 500 ms
   "2915RS001A01L02.FP_PARAM.OpenLoopDelay_Acc" : Int AT %DB5040.DBW138, 500 ms
   "2915RS001A01L02.FP_PARAM.OverRangeDelay_Pre" : Int AT %DB5040.DBW140, 500 ms
   "2915RS001A01L02.FP_PARAM.OverRangeDelay_Acc" : Int AT %DB5040.DBW142, 500 ms
   "2915RS001A01L02.FP_PARAM.AuxLimit_H2_Value" : Real AT %DB5040.DBD144, 500 ms
   "2915RS001A01L02.FP_PARAM.AuxLimit_H1_Value" : Real AT %DB5040.DBD148, 500 ms
   "2915RS001A01L02.FP_PARAM.AuxLimit_L2_Value" : Real AT %DB5040.DBD152, 500 ms
   "2915RS001A01L02.FP_PARAM.AuxLimit_L1_Value" : Real AT %DB5040.DBD156, 500 ms
   "2915RS001A01L02.Unit" : TextRef, internal   // Еденицы измерения При експорте из ECS через скрипт заполняется автоматически, если теги копируются в ручную то требуется задатать свойство Text
   "2915RS001A01L02.Decimals" : TextRef, internal   // Формат отображения При експорте из ECS через скрипт, заполняется автоматически. Если теги копируются в ручную то требуется задатать свойство Text s999999.9
   "2915RS001A01L02.FP_EN.Square" : Bool AT %DB5040.DBX46.0, 500 ms
   "2915RS001A01L02.FP_EN.SquareRoot" : Bool AT %DB5040.DBX46.1, 500 ms
   "2915RS001A01L02.FP_EN.ParentSupress" : Bool AT %DB5040.DBX46.2, 500 ms
   "2915RS001A01L02.FP_EN.ParentSupressUnit" : Bool AT %DB5040.DBX46.3, 500 ms
   "2915RS001A01L02.FP_EN.Force" : Bool AT %DB5040.DBX46.4, 500 ms
   "2915RS001A01L02.FP_EN.Damping" : Bool AT %DB5040.DBX46.5, 500 ms
   "2915RS001A01L02.FP_EN.Gradient_Pos" : Bool AT %DB5040.DBX46.6, 500 ms
   "2915RS001A01L02.FP_EN.Gradient_Neg" : Bool AT %DB5040.DBX46.7, 500 ms
   "2915RS001A01L02.FP_EN.Hysteresis" : Bool AT %DB5040.DBX47.0, 500 ms
   "2915RS001A01L02.FP_EN.Alarm_H3" : Bool AT %DB5040.DBX47.1, 500 ms
   "2915RS001A01L02.FP_EN.Alarm_H2" : Bool AT %DB5040.DBX47.2, 500 ms
   "2915RS001A01L02.FP_EN.Alarm_H1" : Bool AT %DB5040.DBX47.3, 500 ms
   "2915RS001A01L02.FP_EN.Alarm_L1" : Bool AT %DB5040.DBX47.4, 500 ms
   "2915RS001A01L02.FP_EN.Alarm_L2" : Bool AT %DB5040.DBX47.5, 500 ms
   "2915RS001A01L02.FP_EN.Alarm_L3" : Bool AT %DB5040.DBX47.6, 500 ms
   "2915RS001A01L02.FP_EN.AlarmDelay_H3" : Bool AT %DB5040.DBX47.7, 500 ms
   "2915RS001A01L02.FP_EN.AlarmDelay_H2" : Bool AT %DB5040.DBX48.0, 500 ms
   "2915RS001A01L02.FP_EN.AlarmDelay_H1" : Bool AT %DB5040.DBX48.1, 500 ms
   "2915RS001A01L02.FP_EN.AlarmDelay_L1" : Bool AT %DB5040.DBX48.2, 500 ms
   "2915RS001A01L02.FP_EN.AlarmDelay_L2" : Bool AT %DB5040.DBX48.3, 500 ms
   "2915RS001A01L02.FP_EN.AlarmDelay_L3" : Bool AT %DB5040.DBX48.4, 500 ms
   "2915RS001A01L02.FP_EN.ROC_Warn" : Bool AT %DB5040.DBX48.5, 500 ms
   "2915RS001A01L02.FP_EN.U_Range_Warn" : Bool AT %DB5040.DBX48.6, 500 ms
   "2915RS001A01L02.FP_EN.O_Range_Warn" : Bool AT %DB5040.DBX48.7, 500 ms
   "2915RS001A01L02.trend_tag_name" : TextRef, internal   // Еденицы измерения При експорте из ECS через скрипт - заполняется автоматически, если теги копируются в ручную то требуется задатать свойство Text - имя тега для тренда
   "2915RS001A01L02.DQ.AL_H3" : Bool AT %DB5040.DBX16.0, 500 ms
   "2915RS001A01L02.DQ.AL_H2" : Bool AT %DB5040.DBX16.1, 500 ms
   "2915RS001A01L02.DQ.AL_H1" : Bool AT %DB5040.DBX16.2, 500 ms
   "2915RS001A01L02.DQ.AL_L1" : Bool AT %DB5040.DBX16.3, 500 ms
   "2915RS001A01L02.DQ.AL_L2" : Bool AT %DB5040.DBX16.4, 500 ms
   "2915RS001A01L02.DQ.AL_L3" : Bool AT %DB5040.DBX16.5, 500 ms
   "2915RS001A01L02.DQ.SIG_OK" : Bool AT %DB5040.DBX16.6, 500 ms
   "2915RS001A01L02.DQ.LIM_H2" : Bool AT %DB5040.DBX16.7, 500 ms
   "2915RS001A01L02.DQ.LIM_H1" : Bool AT %DB5040.DBX17.0, 500 ms
   "2915RS001A01L02.DQ.LIM_L1" : Bool AT %DB5040.DBX17.1, 500 ms
   "2915RS001A01L02.DQ.LIM_L2" : Bool AT %DB5040.DBX17.2, 500 ms
   "2915RS001A01L02.DQ.GR_P" : Bool AT %DB5040.DBX17.3, 500 ms
   "2915RS001A01L02.DQ.GR_N" : Bool AT %DB5040.DBX17.4, 500 ms
   "2915RS001A01L02.I.IN" : Real AT %DB5040.DBD2, 500 ms
   "2915RS001A01L02.I.SIG_TYPE" : Int AT %DB5040.DBW0, 500 ms
   "2915RS001A01L02.I.FI_BUS" : Byte AT %DB5040.DBB6, 500 ms
   "2915RS001A01L02.DI.U_RANGE" : Bool AT %DB5040.DBX7.0, 500 ms
   "2915RS001A01L02.DI.O_RANGE" : Bool AT %DB5040.DBX7.1, 500 ms
   "2915RS001A01L02.DI.SIG_FAULT" : Bool AT %DB5040.DBX7.2, 500 ms
   "2915RS001A01L02.DI.EnConfig" : Bool AT %DB5040.DBX7.3, 500 ms
   "2915RS001A01L02.DI.AEN" : Bool AT %DB5040.DBX7.4, 500 ms
   "2915RS001A01L02.DI.AL_SUPR" : Bool AT %DB5040.DBX7.5, 500 ms
   "2915RS001A01L02.Q.PV_NORM" : Real AT %DB5040.DBD8, 500 ms
   "2915RS001A01L02.Q.PV_SCAL" : Real AT %DB5040.DBD12, 500 ms
   "2915RS001A01L02.ParentInfo" : TextRef, internal   // Имя родителя для попап окна, вкладка инфо. При експорте из ECS через скрипт заполняется автоматически, если теги копируются в ручную то требуется в ручную задатать свойство Start Value

